(* Logix 5000 project; controller RSL5k_18_Template_noLib Emulate 5570 rev 32.11; software revision 32.02; part 7 of 16 *)
(* tags used below, declared in another part *)
   Inp_CascSP : ALIAS FOR Wrk_PIDE.SPCascade;   // Setpoint in Cascade, Independent PV in Ratio (PVEU)
   Inp_CVPrev : REAL;   // Previous scan CV (CVEU)
   Inp_OvrdCmd : DINT;   // Loop Mode command in Override: 0=None, 1=Man, 2=Auto, 3=Casc, 4=Norm, 5=Start SP Ramp, 6=Stop SP Ramp
   Inp_OvrdSP : REAL;   // Loop Auto Setpoint (SP) in Override (PVEU)
   Inp_OvrdCV : REAL;   // Loop Manual Output (CV) in Override (CVEU)
   Inp_OvrdSPTarget : REAL;   // Override Setpoint Target for SP Ramping ('wizard') (PVEU)
   Inp_OvrdSPRoCLimInc : REAL;   // Override Setting for Setpoint Positive Rate of Change Limit (PVEU/sec)
   Inp_OvrdSPRoCLimDec : REAL;   // Override Setting for Setpoint Negative Rate of Change Limit (PVEU/sec)
   Inp_Reset : BOOL;   // 1=Reset latched Alarms
   Cfg_HasRatio : ALIAS FOR Wrk_PIDE.UseRatio;   // 1=Casc Loop Mode is Ratio, 0=Casc Loop Mode is Cascade
   Cfg_HasCasc : ALIAS FOR Wrk_PIDE.AllowCasRat;   // 1=Enable the loop to be placed into cascade/ratio mode
   Cfg_HasAuto : BOOL;   // 1=Enable the loop to be placed into automatic mode
   Cfg_HasMan : BOOL;   // 1=Enable the loop to be placed into manual mode
   Cfg_LockLM : BOOL;   // Lock Loop Mode: 0=not locked, 1=locked in Normal mode (see Cfg_NormLM)
   Cfg_HasMoreObj : BOOL;   // 1=Tells HMI an object with more info is available
   Cfg_OvrdIntlk : BOOL;   // 1=Override ignores Bypassable Intlk; 0=always use Intlk
   Cfg_NormLM : DINT;   // Normal Loop Mode 0=Disable Normal selection, 1=Man, 2=Auto, 3=Casc
   Cfg_PwrupLM : DINT;   // Powerup Loop Mode 0=No change (last), 1=Man (w/ CV), 2=Auto (w/ SP), 3=Casc, 4=Normal
   Cfg_SPFailSPAct : DINT;   // SP Fail Setpoint Action: 1=hold last good, 2=use Cfg_IntlkSP, 3=set SP to curr. PV
   Cfg_PVFailCVAct : DINT;   // PV Fail CV Action: 1=hold last good, 2=use Cfg_IntlkCV
   Cfg_CVFailCVAct : DINT;   // CV Fail CV Action: 1=hold last good, 2=use Cfg_IntlkCV
   Cfg_PVDecPlcs : DINT;   // Number of decimal places for display of PV / SP
   Cfg_CVDecPlcs : DINT;   // Number of decimal places for display of CV
   Cfg_MaxSPRoCInc : REAL;   // Maximum allowed Setpoint Positive Rate of Change Limit (PVEU/sec)
   Cfg_MaxSPRoCDec : REAL;   // Maximum allowed Setpoint Negative Rate of Change Limit (PVEU/sec)
   Cfg_CVEUMin : REAL;   // CV Engineering Units Minimum Value (CVEU)
   Cfg_CVEUMax : REAL;   // CV Engineering Units Maximum Value (CVEU)
   Cfg_PGain : ALIAS FOR Wrk_PIDE.PGain;   // Proportional (independent) or Loop (dependent) Gain (unitless)
   Cfg_IGain : ALIAS FOR Wrk_PIDE.IGain;   // Integral Gain (1/min independent or min/repeat dependent)
   Cfg_DGain : ALIAS FOR Wrk_PIDE.DGain;   // Derivative Gain (min)
   Cfg_ZCDB : ALIAS FOR Wrk_PIDE.ZCDeadband;   // Normal Zero Crossing Deadband (PVEU)
   Cfg_CVRoCLim : REAL;   // CV Rate of Change Limit (CVEU/sec)
   Cfg_IntlkCV : REAL;   // CV Value to use with Interlock / Bad Value CV action (CVEU)
   Cfg_PwrupSP : REAL;   // Loop SP on powerup, used if Cfg_PwrupLM = 1 (Manual) or 2 (Auto) (PVEU)
   Cfg_PwrupCV : REAL;   // Loop CV on powerup, used if Cfg_PwrupLM <> 0 (none) (CVEU)
   Cfg_HiHiDevDB : REAL;   // High-High Devation Status Deadband (PVEU)
   Cfg_HiDevDB : REAL;   // High Devation Status Deadband (PVEU)
   Cfg_LoDevDB : REAL;   // Low Devation Status Deadband (PVEU)
   Cfg_LoLoDevDB : REAL;   // Low-Low Devation Status Deadband (PVEU)
   Cfg_OperKeep : SINT;   // Oper keeps control: .0=Loop Mode .1=CV .2=SP, .3=Ratio
   Cfg_ProgKeep : SINT;   // Prog keeps control: .0=Loop Mode .1=CV .2=SP, .3=Ratio
   Cfg_ExtKeep : SINT;   // Ext keeps control: .0=Loop Mode .1=CV .2=SP, .3=Ratio
   PSet_SP : REAL;   // Program Setting for Setpoint (loop Auto) (PVEU)
   PSet_SPRoCLimInc : REAL;   // Program Setting for Setpoint Rate of Change Limit Increasing (PVEU/sec)
   PSet_SPRoCLimDec : REAL;   // Program Setting for Setpoint Rate of Change Limit Decreasing (PVEU/sec)
   PSet_SPTarget : REAL;   // Program Setting for Setpoint Ramp Target (endpoint, for ramp wizard) (PVEU)
   PSet_CV : REAL;   // Program Setting for Controlled Variable (loop Manual) (CVEU)
   PSet_Owner : DINT;   // Program Owner Request ID (non-zero) or Release (zero)
   XSet_SP : REAL;   // External Setting for Setpoint (loop Auto) (PVEU)
   XSet_SPRoCLimInc : REAL;   // External Setting for Setpoint Rate of Change Limit Increasing (PVEU/sec)
   XSet_SPRoCLimDec : REAL;   // External Setting for Setpoint Rate of Change Limit Decreasing (PVEU/sec)
   XSet_SPTarget : REAL;   // External Setting for Setpoint Ramp Target (endpoint, for ramp wizard) (PVEU)
   XSet_CV : REAL;   // External Setting for Controlled Variable (loop Manual) (CVEU)
   PCmd_Casc : BOOL;   // Program Command to select Cascade / Ratio Loop Mode
   PCmd_Auto : BOOL;   // Program Command to select Automatic Loop Mode
   PCmd_Man : BOOL;   // Program Command to select Manual Loop Mode
   PCmd_NormLM : BOOL;   // Operator Command to select Normal Loop Mode (see Cfg_NormLM)
   PCmd_SPRampStart : BOOL;   // Program Command to initiate SP ramping
   PCmd_SPRampStop : BOOL;   // Program Command to stop SP ramping
   PCmd_Reset : BOOL;   // Program Command to Reset all Alarms requiring Reset
   XCmd_Casc : BOOL;   // External Command to select Cascade / Ratio control
   XCmd_Auto : BOOL;   // External Command to select Automatic control
   XCmd_Man : BOOL;   // External Command to select Manual control
   XCmd_NormLM : BOOL;   // External Command to select Normal Loop Mode (see Cfg_NormLM)
   XCmd_SPRampStart : BOOL;   // External Command to initiate SP ramping
   XCmd_SPRampStop : BOOL;   // External Command to stop SP ramping
   XCmd_Reset : BOOL;   // External Command to Reset all Alarms requiring Reset
   Val_Ratio : ALIAS FOR Wrk_PIDE.Ratio;   // Value of Loop Ratio (unitless)
   Val_SPSet : REAL;   // Value of selected SP (before clamping and ramping) (PVEU)
   Val_SP : ALIAS FOR Wrk_PIDE.SP;   // Value of SP being used (after ramping and clamping (PVEU)
   Val_SPTarget : REAL;   // Accepted Setting for Setpoint Ramp Target (endpoint, for ramp wizard) (PVEU)
   Val_CVSet : REAL;   // Value of selected CV (before clamping and ramping) (CVEU)
   Val_CVOut : REAL;   // Value of CV Output (after ramping and clamping (CVEU)
   Val_Owner : DINT;   // Current Object Owner ID (0=not owned)
   Sts_PVBad : BOOL;   // 1=PV Value, comms, quality or EU Limitis Bad
   Sts_Bypass : BOOL;   // 1=Bypassable Interlocks are Bypassed
   Sts_BypActive : BOOL;   // 1=Bypassing Active (Bypassed or Maintenance)
   Nrdy_OoS : BOOL;   // 1=Device Not Ready: Out of Service
   Sts_MaintByp : BOOL;   // 1=Device has a Maintenance Bypass function active
   Err_CVEU : BOOL;   // 1=Error in Config: CV EU Max/Min Invalid
   Sts_OoS : ALIAS FOR CmdSrc.Sts_OoS;
   Sts_Maint : ALIAS FOR CmdSrc.Sts_Maint;
   Sts_Ovrd : ALIAS FOR CmdSrc.Sts_Ovrd;
   Sts_Ext : ALIAS FOR CmdSrc.Sts_Ext;
   Sts_Prog : ALIAS FOR CmdSrc.Sts_Prog;
   Sts_Oper : ALIAS FOR CmdSrc.Sts_Oper;
   Sts_RdyAck : BOOL;   // 1=An alarm is ready to be acknowledged
   P_PIDE : BOOL;   // Unique Parameter Name for auto - discovery
   CmdSrc : P_CmdSrc;   // Control / Command Source Selection
   Fail : P_Alarm;   // Loop (SP, PV or CV) Failure Alarm
   IntlkTrip : P_Alarm;   // Interlock Trip Alarm
   Cfg_Tag : STRING_20;   // Tagname displayed on HMI
   Cfg_Label : STRING_20;   // Label for graphic symbol displayed on HMI
   Cfg_Desc : STRING_40;   // Description displayed on HMI
   Wrk_Bypass : BOOL;   // Internal Bypassable Interlocks are Bypassed flag
   Cfg_PVEU : STRING_8;   // PV / Setpoint Engineering Units displayed on HMI
   Wrk_ProgKeepONS : SINT;   // Program Keep one-shot stores
   Wrk_OperKeepONS : SINT;   // Operator Keep one-shot stores
   Wrk_ExtKeepONS : SINT;   // External Keep one-shot stores
   LoLoDev : P_Alarm;   // Low-Low Deviation Alarm
   LoDev : P_Alarm;   // Low Deviation Alarm
   HiDev : P_Alarm;   // High Deviation Alarm
   HiHiDev : P_Alarm;   // High-High Deviation Alarm
   Cfg_CVEU : STRING_8;   // CV Engineering Units displayed on HMI
   Wrk_Casc : BOOL;   // Internal Loop Mode latch: Cascade selected
   Wrk_Auto : BOOL;   // Internal Loop Mode latch: 1=Auto selected
   Wrk_Man : BOOL;   // Internal Loop Mode latch: Manual selected
   HMI_Type : STRING_16;   // Must contain AOI name, used for HMI and Information S/W
   Wrk_IntlkTripShed : BOOL;   // Shed Latch for Interlock Not OK
   Wrk_PVFailShed : BOOL;   // Shed Latch for PV Failure
   Wrk_SPFailShed : BOOL;   // Shed Latch for SP Failure
   Wrk_CVFailShed : BOOL;   // Shed Latch for CV Failure
   Wrk_ShedMan : BOOL;   // A shed condition is forcing Loop Mode to Manual
   Wrk_ShedAuto : BOOL;   // A shed condition is forcing Loop Mode to Auto or Manual
   Cfg_CVNavTag : STRING_NavTag;   // Tagname for destination of CV Navigation button
   Cfg_PVNavTag : STRING_NavTag;   // Tagname for destination of PV Navigation button
   Cfg_CascSPNavTag : STRING_NavTag;   // Tagname for destination of Cascade SP Navigation button
   HMI_Lib : STRING_12;   // Display Library for Faceplate call-up
   Wrk_PIDE : PID_ENHANCED;   // Built-in controller PID algorithm
   Cfg_Area : STRING_Area;   // Process Area for security
   Wrk_Autotune : PIDE_AUTOTUNE;   // Autotune tag associated with built-in PID algorithm
   HMI_HasAutotune : BOOL;   // 1=P_PIDE_Only AOI has been modified to include Autotune par. on PIDE block
   OCmd_ResetAckAll : BOOL;   // Operator Command to Reset all Alarms and latched Shed conditions
   OCmd_Reset : BOOL;   // Operator Command to Reset all Alarms requiring Reset
   MCmd_Check : BOOL;   // Maintenance Command to Check (not bypass) all Interlocks
   MCmd_Bypass : BOOL;   // Maintenance Command to Bypass all Bypassable Interlocks
   OCmd_SPRampStop : BOOL;   // Operator Command to stop SP ramping
   OCmd_SPRampStart : BOOL;   // Operator Command to initiate SP ramping
   OCmd_NormLM : BOOL;   // Operator Command to select Normal Loop Mode (see Cfg_NormLM)
   OCmd_Man : BOOL;   // Operator Command to select Manual control
   OCmd_Auto : BOOL;   // Operator Command to select Automatic control
   OCmd_Casc : BOOL;   // Operator Command to select Cascade / Ratio control
   OSet_CV : REAL;   // Operator Setting for Controlled Variable (loop Manual) (CVEU)
   OSet_SPTarget : REAL;   // Operator Setting for Setpoint Ramp Target (endpoint, for ramp wizard) (PVEU)
   OSet_SPRoCLimDec : REAL;   // Operator Setting for Setpoint Rate of Change Limit Decreasing (PVEU/sec)
   OSet_SPRoCLimInc : REAL;   // Operator Setting for Setpoint Rate of Change Limit Increasing (PVEU/sec)
   OSet_SP : REAL;   // Operator Setting for Setpoint (loop Auto) (PVEU)
   Wrk_ExtHas : SINT;   // External owns: .0=LM, .1=CV, .2=SP, .3=Ratio
   Wrk_ProgHas : SINT;   // Program owns: .0=LM, .1=CV, .2=SP, .3=Ratio
   Wrk_OperHas : SINT;   // Operator owns: .0=LM, .1=CV, .2=SP, .3=Ratio
   MRdy_Check : BOOL;   // 1=Ready for MCmd_Check (enables HMI button)
   MRdy_Bypass : BOOL;   // 1=Ready for MCmd_Bypass (enables HMI button)
   Wrk_Init : BOOL;   // 1=AOI has been initialized
(* P_PIDE, continued *)

ROUTINE Logic   (* ladder *)
// Normal Scan: control PID Loop
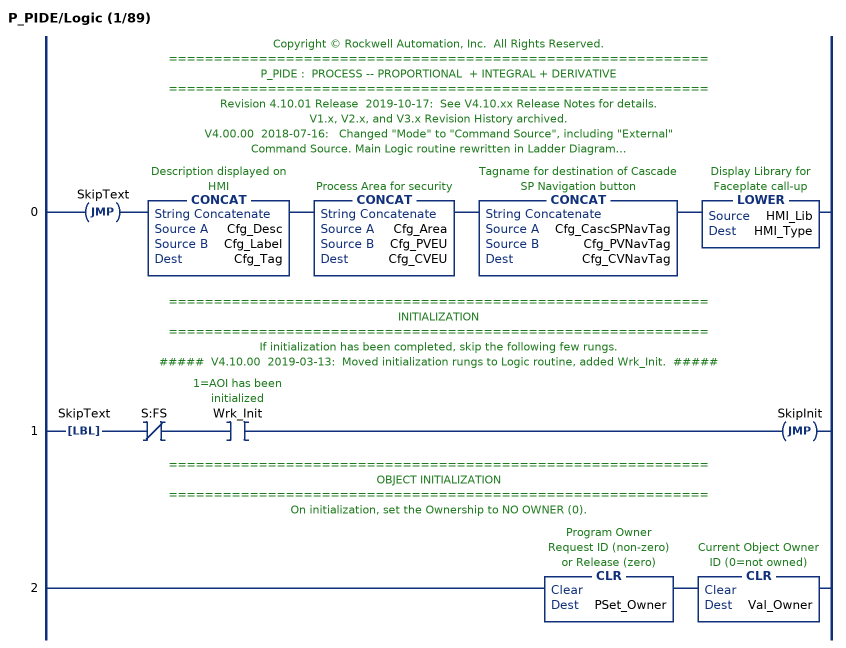
   // Copyright © Rockwell Automation, Inc.  All Rights Reserved.
   // ============================================================
   // P_PIDE :  PROCESS -- PROPORTIONAL  + INTEGRAL + DERIVATIVE
   // ============================================================
   // Revision 4.10.01 Release  2019-10-17:  See V4.10.xx Release Notes for details.
   // V1.x, V2.x, and V3.x Revision History archived.
   // V4.00.00  2018-07-16:   Changed "Mode" to "Command Source", including "External"
   // Command Source. Main Logic routine rewritten in Ladder Diagram.
   // Changed Inf_ items to HMI_, and added Cfg_Area for security.
   // Added notify and unack count rollup for connected objects.
   // Deleted Cfg_PCmdClear.  All Program Commands are now self-clearing.
   // Aligned ready bit naming with command bit names.
   // All OCmds/MCmds and ORdys/MRdys are now Local Tags.
   // Added Sts_RdyAck and Sts_ResetReqd for use by external objects.
   // Added SP Ramping and Ramp Wizard.  Added capability to have CV range
   // other than 0 to 100%.  Added Shed options.  Added Normal Loop Mode, locking
   // of Loop Mode. Added Oper / Prog / Ext "Keep" for Loop Mode, CV, SP, Ratio.
   // V4.00.01  2018-08-29:  Updated Override Command Source operation and description of Inp_OvrdCmd.
   // V4.00.02  2018-12-10:  Modified handling of CV I/O Fault, CV Fail and Shed configurations.
   // Corrected handling of configured execution interval.
   // V4.10.00  2019-03-13:  Changed availability to use input availability from interlocks.
   // Corrected parameter and local tag descriptions and external access.
   // Added Cfg_HasMoreObj. Updated to P_CmdSrc V4.10.00.
   // Moved initialization rungs to Logic routine, added Wrk_Init to correct
   // locking of Autotune tag on online instance creation.
   // Corrected overwriting of user SP Rate of Change limits by SP ramp wizard.
   // V4.10.01  2019-10-17:  Corrected clamping of CV, Ratio settings in Manual.
   // Corrected determination of Val_CVSet based on CV Init status.
   // Corrected generation of Sts_PVBad. Corrected CV Rate of Change Limiting.
   // Modified Interlock function to use PIDE manual CV instead of override CV, to get CV ramping.
   // Corrected SP ramp increasing. Modified Cascade/Ratio logic to include SP rate limiting.
   // ============================================================
   // This Instruction is used to provide PID (Proportional + Integral +
   // Derivative) feedback loop control and provides:
   // *  Prog, Oper, and Ext entry of Auto loop mode Setpoint in Engineering Units
   // *  Prog, Oper, and Ext. entry of Setpoint Target and Ramp Time and
   // command to trigger a Setpoint Ramp ("SP Ramp Wizard")
   // *  Prog, Oper, and Ext. entry of Manual loop mode Controlled Variable (CV) in Percent
   // *  Clamping (in EU) and ramping (in EU/sec) of Setpoint at specified limits
   // (separate increase and decrease rate of change limits).
   // *  Clamping (in CVEU) and ramping (in CVEU/sec) of CV at specified limits
   // (separate increase and decrease rate of change limits).
   // *  CV in Engineering Units (CVEU) for use as Cascade Setpoint for a secondary loop\
   // plus scaling to Raw units for use with non-scaling I/O card
   // *  Reverse or Direct control action    *  Feedforward input
   // *  Velocity (difference) PID form (with inputs for "Previous" CV and FF)
   // *  Option for Derivative action based on change in Error or change in PV
   // *  Option for Proportional action based on Error or PV
   // *  Monitoring of Interlock conditions which cause output to shed
   // *  Configurable shed to HOLD or to configured SAFE value, shed SP to current PV.
   // *  Monitoring of I/O communication faults
   // *  Alarms for Interlock Trip, Loop Failure, High-High Deviation, High Deviation,
   // Low Deviation and Low-Low Deviation from Setpoint
   // *  Operation from Hand, Maintenance, Override, External Program and Operator command sources
   // *  Full loop control (Cascade, Auto with Setpoint, Manual with CV) available in Override
   // *  "Available" status for use by automation logic to know whether loop
   //       can be controlled via Program commands / settings from other objects.
   // Command Sources are arbitrated by a P_CmdSrc Add-On Instruction instance.
   // Command Sources: Operator, Program, External, Override, Maintenance,
   // Out of Service, Hand.  Alarms are provided by P_Alarm Add-On Instruction instances.
   // ============================================================
   // SHOW LOCAL STRINGS
   // ============================================================
   // The STRINGs containing the text associated with each instance of this
   // instruction cannot be Input or Output Parameters, because STRINGs are not
   //  'atomic' types. (Inputs and Outputs must be SINT, INT, DINT, REAL, or BOOL.)
   // In order to make it easier to find and configure these STRINGs, this rung
   // was added.  THE JMP (and the LBL on the following rung)
   // MUST NOT BE REMOVED!!!
   // To view the STRINGs, go to the instruction instance (in LD or FBD), RIGHT-click
   // to bring up the context menu and select "Open Instruction Logic".
   // This rung will appear with the STRING values for the selected instance.
   // You may double-click the STRING values here to modify them as well.
   // #####  V4.00.00  2018-07-16:  Added string for Cfg_Area, renamed Inf_* to HMI_*.  #####
   0: JMP(SkipText)CONCAT(Cfg_Desc,Cfg_Label,Cfg_Tag)CONCAT(Cfg_Area,Cfg_PVEU,Cfg_CVEU)CONCAT(Cfg_CascSPNavTag,Cfg_PVNavTag,Cfg_CVNavTag)LOWER(HMI_Lib,HMI_Type);
   // ============================================================
   // INITIALIZATION
   // ============================================================
   // If initialization has been completed, skip the following few rungs.
   // #####  V4.10.00  2019-03-13:  Moved initialization rungs to Logic routine, added Wrk_Init.  #####
   1: LBL(SkipText)XIO(S:FS)XIC(Wrk_Init)JMP(SkipInit);
   // ============================================================
   // OBJECT INITIALIZATION
   // ============================================================
   // On initialization, set the Ownership to NO OWNER (0).
   2: CLR(PSet_Owner)CLR(Val_Owner);
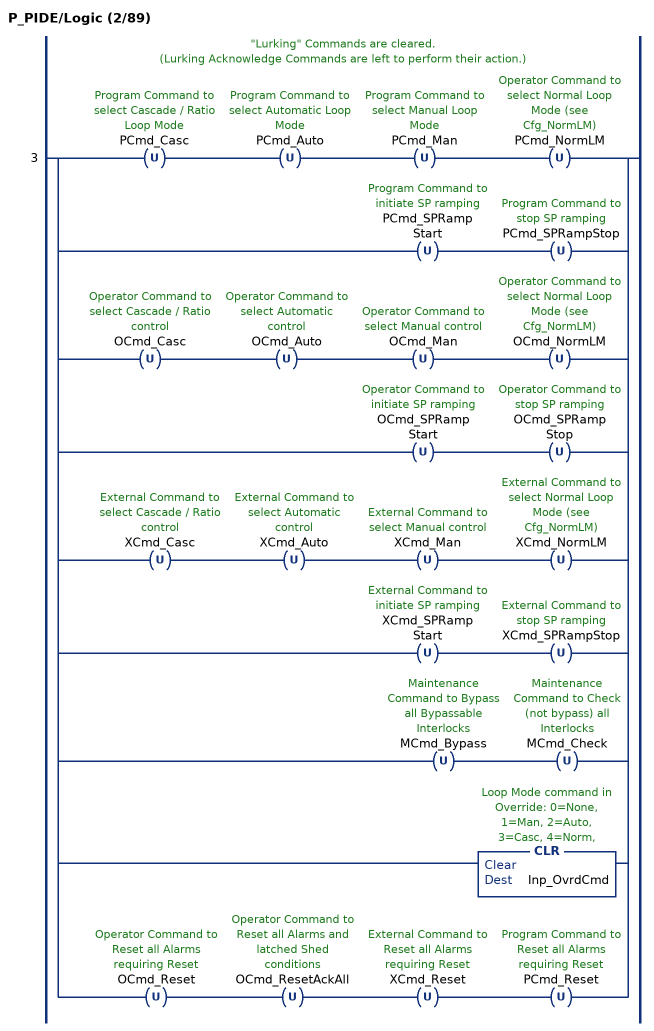
   // "Lurking" Commands are cleared.
   // (Lurking Acknowledge Commands are left to perform their action.)
   3: [OTU(PCmd_Casc) OTU(PCmd_Auto) OTU(PCmd_Man) OTU(PCmd_NormLM) ,OTU(PCmd_SPRampStart) OTU(PCmd_SPRampStop) ,OTU(OCmd_Casc) OTU(OCmd_Auto) OTU(OCmd_Man) OTU(OCmd_NormLM) ,OTU(OCmd_SPRampStart) OTU(OCmd_SPRampStop) ,OTU(XCmd_Casc) OTU(XCmd_Auto) OTU(XCmd_Man) OTU(XCmd_NormLM) ,OTU(XCmd_SPRampStart) OTU(XCmd_SPRampStop) ,OTU(MCmd_Bypass) OTU(MCmd_Check) ,CLR(Inp_OvrdCmd) ,OTU(OCmd_Reset) OTU(OCmd_ResetAckAll) OTU(XCmd_Reset) OTU(PCmd_Reset) ];
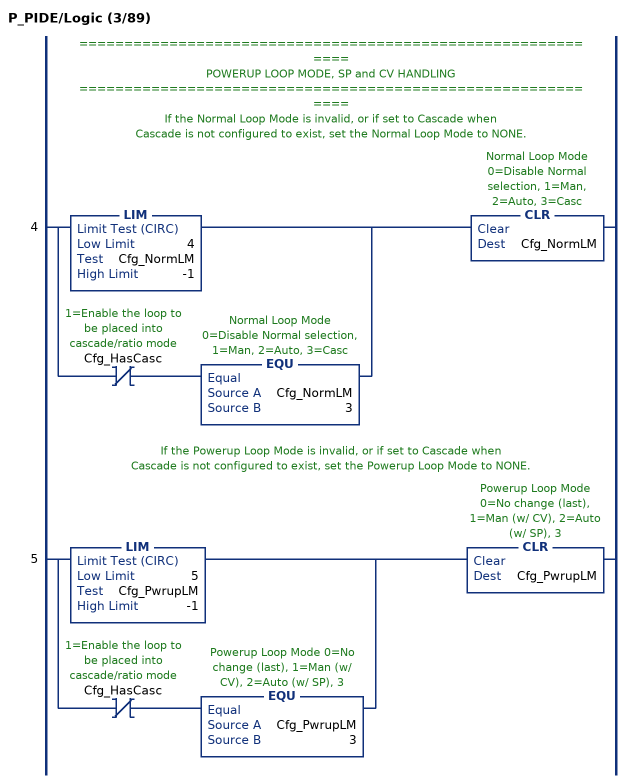
   // ============================================================
   // POWERUP LOOP MODE, SP and CV HANDLING
   // ============================================================
   // If the Normal Loop Mode is invalid, or if set to Cascade when
   // Cascade is not configured to exist, set the Normal Loop Mode to NONE.
   4: [LIM(4,Cfg_NormLM,-1) ,XIO(Cfg_HasCasc) EQU(Cfg_NormLM,3) ]CLR(Cfg_NormLM);
   // If the Powerup Loop Mode is invalid, or if set to Cascade when
   // Cascade is not configured to exist, set the Powerup Loop Mode to NONE.
   5: [LIM(5,Cfg_PwrupLM,-1) ,XIO(Cfg_HasCasc) EQU(Cfg_PwrupLM,3) ]CLR(Cfg_PwrupLM);
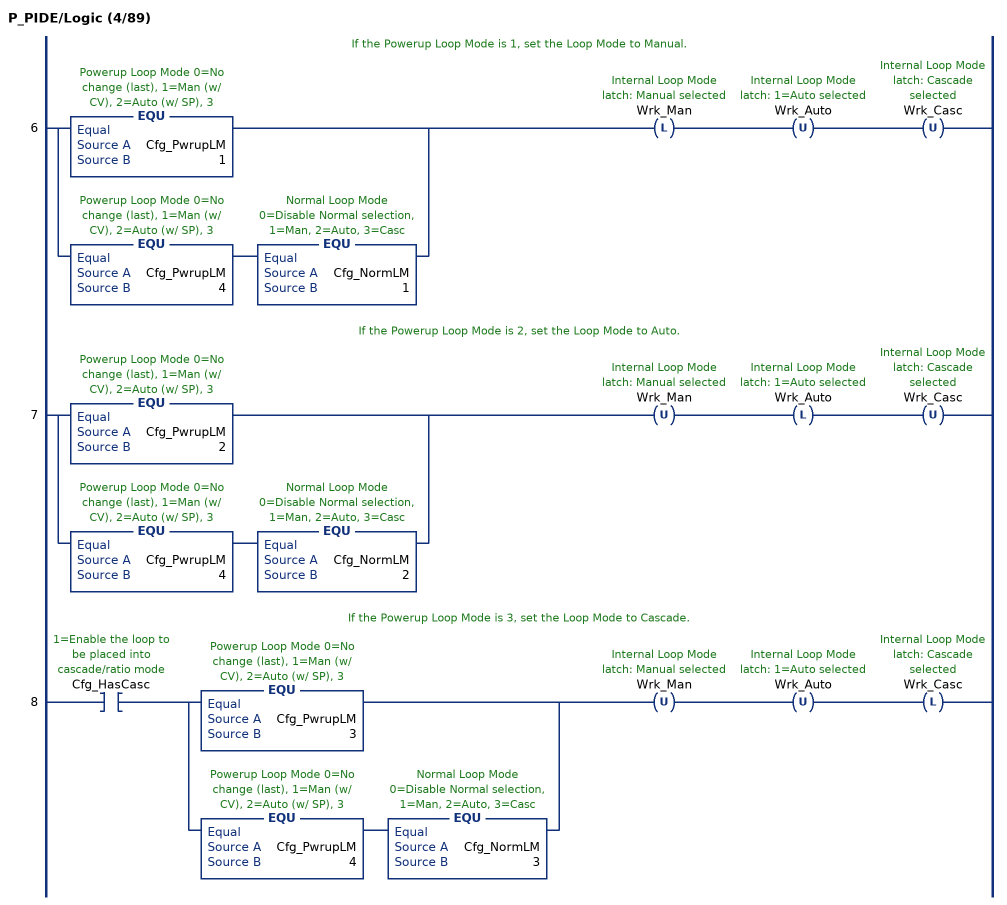
   // If the Powerup Loop Mode is 1, set the Loop Mode to Manual.
   6: [EQU(Cfg_PwrupLM,1) ,EQU(Cfg_PwrupLM,4) EQU(Cfg_NormLM,1) ]OTL(Wrk_Man)OTU(Wrk_Auto)OTU(Wrk_Casc);
   // If the Powerup Loop Mode is 2, set the Loop Mode to Auto.
   7: [EQU(Cfg_PwrupLM,2) ,EQU(Cfg_PwrupLM,4) EQU(Cfg_NormLM,2) ]OTU(Wrk_Man)OTL(Wrk_Auto)OTU(Wrk_Casc);
   // If the Powerup Loop Mode is 3, set the Loop Mode to Cascade.
   8: XIC(Cfg_HasCasc)[EQU(Cfg_PwrupLM,3) ,EQU(Cfg_PwrupLM,4) EQU(Cfg_NormLM,3) ]OTU(Wrk_Man)OTU(Wrk_Auto)OTL(Wrk_Casc);
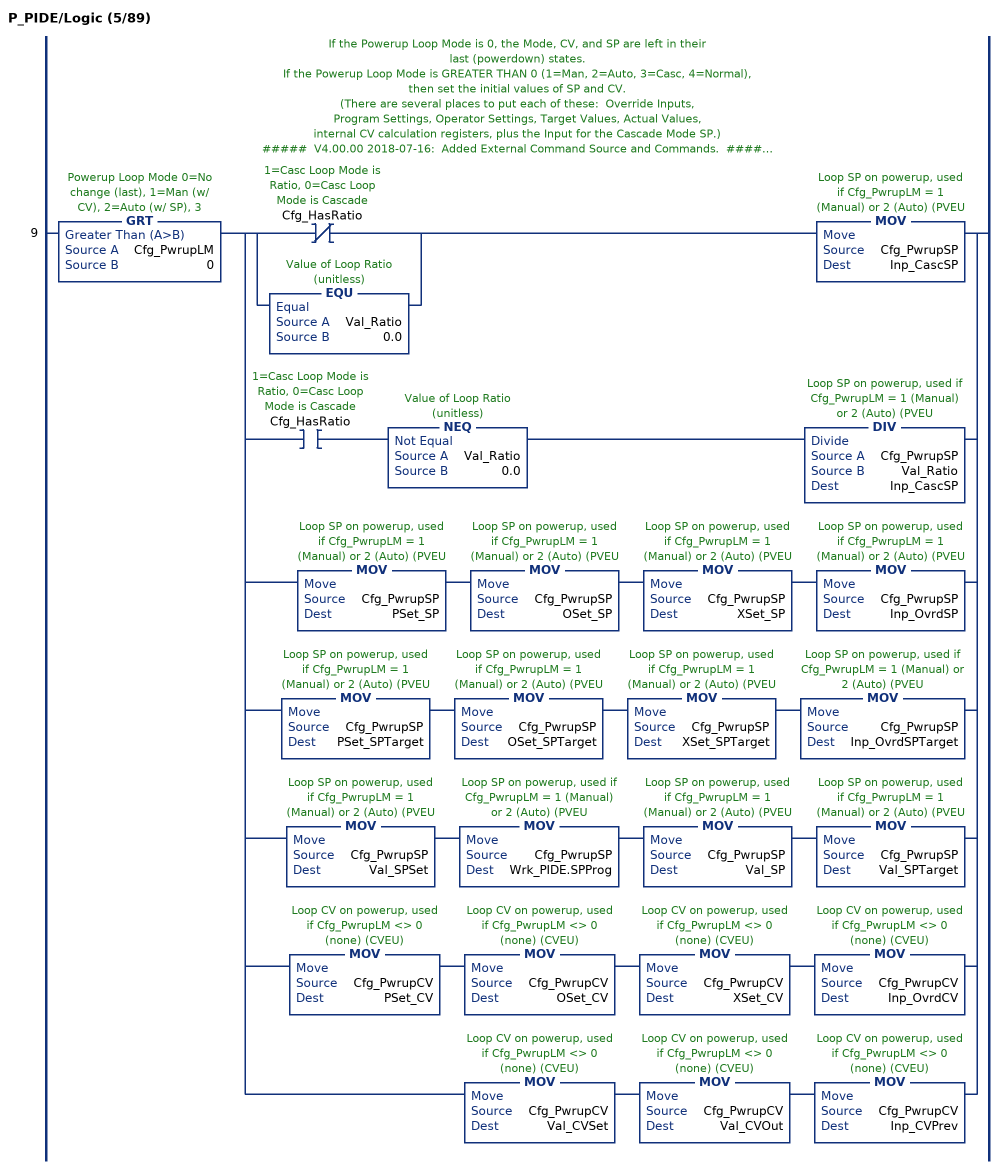
   // If the Powerup Loop Mode is 0, the Mode, CV, and SP are left in their
   // last (powerdown) states.
   // If the Powerup Loop Mode is GREATER THAN 0 (1=Man, 2=Auto, 3=Casc, 4=Normal),
   // then set the initial values of SP and CV.
   // (There are several places to put each of these:  Override Inputs,
   // Program Settings, Operator Settings, Target Values, Actual Values,
   // internal CV calculation registers, plus the Input for the Cascade Mode SP.)
   // #####  V4.00.00 2018-07-16:  Added External Command Source and Commands.  #####
   // #####  V4.00.02  2018-12-10:  Modified handling of CV Init, CV I/O Fault, and Powerup CV.  #####
   9: GRT(Cfg_PwrupLM,0)[[[XIO(Cfg_HasRatio) ,EQU(Val_Ratio,0.0) ] MOV(Cfg_PwrupSP,Inp_CascSP) ,XIC(Cfg_HasRatio) NEQ(Val_Ratio,0.0) DIV(Cfg_PwrupSP,Val_Ratio,Inp_CascSP) ] ,MOV(Cfg_PwrupSP,PSet_SP) MOV(Cfg_PwrupSP,OSet_SP) MOV(Cfg_PwrupSP,XSet_SP) MOV(Cfg_PwrupSP,Inp_OvrdSP) ,MOV(Cfg_PwrupSP,PSet_SPTarget) MOV(Cfg_PwrupSP,OSet_SPTarget) MOV(Cfg_PwrupSP,XSet_SPTarget) MOV(Cfg_PwrupSP,Inp_OvrdSPTarget) ,MOV(Cfg_PwrupSP,Val_SPSet) MOV(Cfg_PwrupSP,Wrk_PIDE.SPProg) MOV(Cfg_PwrupSP,Val_SP) MOV(Cfg_PwrupSP,Val_SPTarget) ,MOV(Cfg_PwrupCV,PSet_CV) MOV(Cfg_PwrupCV,OSet_CV) MOV(Cfg_PwrupCV,XSet_CV) MOV(Cfg_PwrupCV,Inp_OvrdCV) ,MOV(Cfg_PwrupCV,Val_CVSet) MOV(Cfg_PwrupCV,Val_CVOut) MOV(Cfg_PwrupCV,Inp_CVPrev) ];
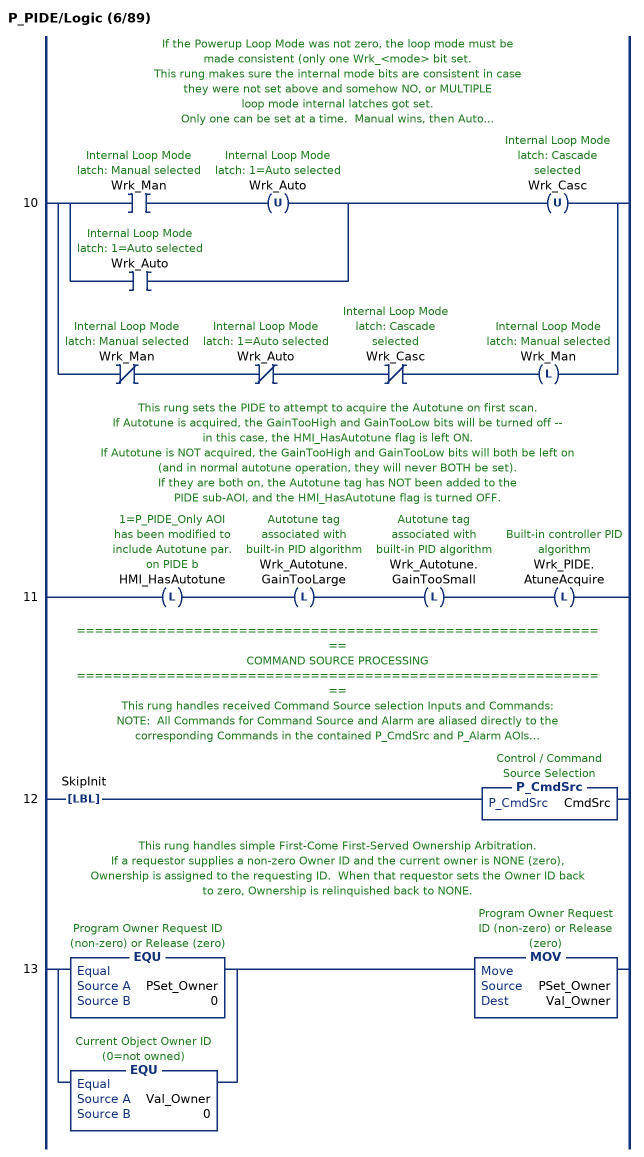
   // If the Powerup Loop Mode was not zero, the loop mode must be
   // made consistent (only one Wrk_<mode> bit set.
   // This rung makes sure the internal mode bits are consistent in case
   // they were not set above and somehow NO, or MULTIPLE
   // loop mode internal latches got set.
   // Only one can be set at a time.  Manual wins, then Auto...
   10: [[XIC(Wrk_Man) OTU(Wrk_Auto) ,XIC(Wrk_Auto) ] OTU(Wrk_Casc) ,XIO(Wrk_Man) XIO(Wrk_Auto) XIO(Wrk_Casc) OTL(Wrk_Man) ];
   // This rung sets the PIDE to attempt to acquire the Autotune on first scan.
   // If Autotune is acquired, the GainTooHigh and GainTooLow bits will be turned off --
   // in this case, the HMI_HasAutotune flag is left ON.
   // If Autotune is NOT acquired, the GainTooHigh and GainTooLow bits will both be left on
   // (and in normal autotune operation, they will never BOTH be set).
   // If they are both on, the Autotune tag has NOT been added to the
   // PIDE sub-AOI, and the HMI_HasAutotune flag is turned OFF.
   11: OTL(HMI_HasAutotune)OTL(Wrk_Autotune.GainTooLarge)OTL(Wrk_Autotune.GainTooSmall)OTL(Wrk_PIDE.AtuneAcquire);
   // ============================================================
   // COMMAND SOURCE PROCESSING
   // ============================================================
   // This rung handles received Command Source selection Inputs and Commands:
   // NOTE:  All Commands for Command Source and Alarm are aliased directly to the
   // corresponding Commands in the contained P_CmdSrc and P_Alarm AOIs.
   // #####  V4.00.00  2018-07-16:  Changed P_Mode to P_CmdSrc.  #####
   // #####  V4.10.00  2019-03-13:  Moved initialization rungs to Logic routine, added Wrk_Init. Added LBL here.  #####
   12: LBL(SkipInit)P_CmdSrc(CmdSrc);
   // This rung handles simple First-Come First-Served Ownership Arbitration.
   // If a requestor supplies a non-zero Owner ID and the current owner is NONE (zero),
   // Ownership is assigned to the requesting ID.  When that requestor sets the Owner ID back
   // to zero, Ownership is relinquished back to NONE.
   13: [EQU(PSet_Owner,0) ,EQU(Val_Owner,0) ]MOV(PSet_Owner,Val_Owner);
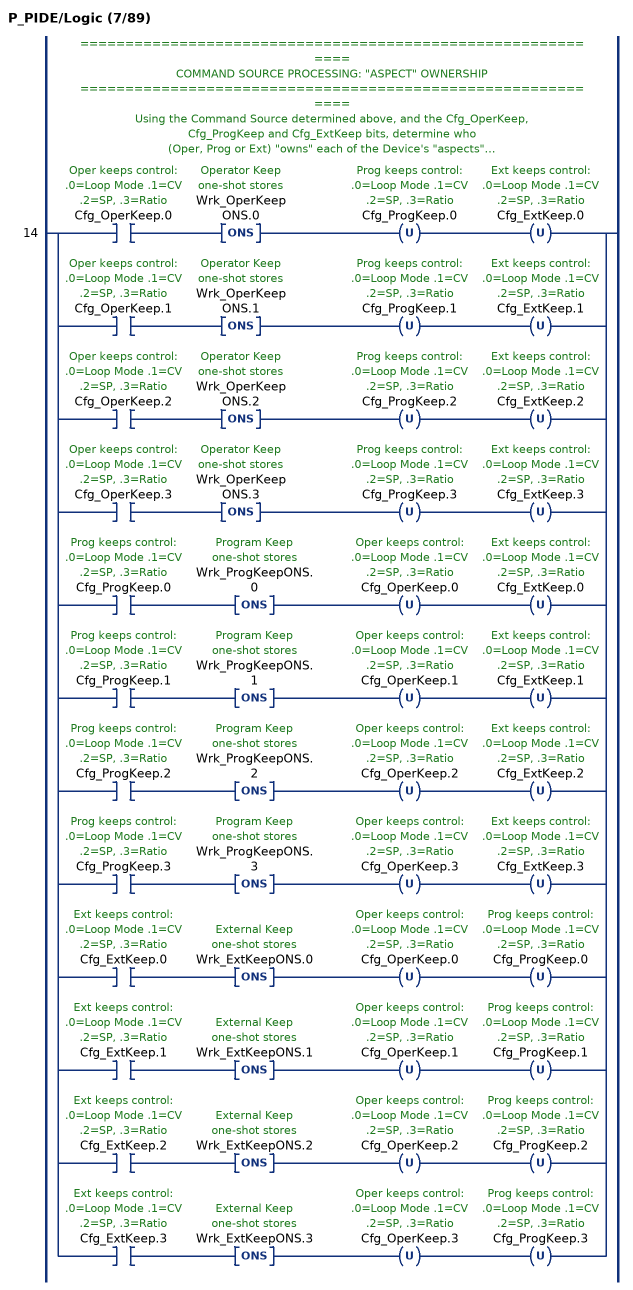
   // ============================================================
   // COMMAND SOURCE PROCESSING: "ASPECT" OWNERSHIP
   // ============================================================
   // Using the Command Source determined above, and the Cfg_OperKeep,
   // Cfg_ProgKeep and Cfg_ExtKeep bits, determine who
   // (Oper, Prog or Ext) "owns" each of the Device's "aspects":
   // Loop Mode (bit .0), Controlled Variable (CV, the output, bit .1),
   // Setpoint (SP, bit .2), and Ratio (bit .3).
   // The bits within Cfg_OperKeep, Cfg_ProgKeep and Cfg_ExtKeep determine
   // which "aspects" (sub-functions of this AOI) are retained by the Operator,
   // by the Program, or by the External command source when either of the
   // other command sources is selected.
   // All aspects (functions) may be "kept" (basically locking the Oper/Prog/Ext
   // selections, rendering the Command Source selection moot.
   // (You get to explain how it works to your operators!!!).
   // However, it is NOT allowed to have any given aspect "kept" by more than
   // one source.  This rung ensures that no aspect is "kept" by multiple sources.
   // #####  V4.00.00  2018-07-16:  Using P_CmdSrc, added External command source.  #####
   14: [XIC(Cfg_OperKeep.0) ONS(Wrk_OperKeepONS.0) OTU(Cfg_ProgKeep.0) OTU(Cfg_ExtKeep.0) ,XIC(Cfg_OperKeep.1) ONS(Wrk_OperKeepONS.1) OTU(Cfg_ProgKeep.1) OTU(Cfg_ExtKeep.1) ,XIC(Cfg_OperKeep.2) ONS(Wrk_OperKeepONS.2) OTU(Cfg_ProgKeep.2) OTU(Cfg_ExtKeep.2) ,XIC(Cfg_OperKeep.3) ONS(Wrk_OperKeepONS.3) OTU(Cfg_ProgKeep.3) OTU(Cfg_ExtKeep.3) ,XIC(Cfg_ProgKeep.0) ONS(Wrk_ProgKeepONS.0) OTU(Cfg_OperKeep.0) OTU(Cfg_ExtKeep.0) ,XIC(Cfg_ProgKeep.1) ONS(Wrk_ProgKeepONS.1) OTU(Cfg_OperKeep.1) OTU(Cfg_ExtKeep.1) ,XIC(Cfg_ProgKeep.2) ONS(Wrk_ProgKeepONS.2) OTU(Cfg_OperKeep.2) OTU(Cfg_ExtKeep.2) ,XIC(Cfg_ProgKeep.3) ONS(Wrk_ProgKeepONS.3) OTU(Cfg_OperKeep.3) OTU(Cfg_ExtKeep.3) ,XIC(Cfg_ExtKeep.0) ONS(Wrk_ExtKeepONS.0) OTU(Cfg_OperKeep.0) OTU(Cfg_ProgKeep.0) ,XIC(Cfg_ExtKeep.1) ONS(Wrk_ExtKeepONS.1) OTU(Cfg_OperKeep.1) OTU(Cfg_ProgKeep.1) ,XIC(Cfg_ExtKeep.2) ONS(Wrk_ExtKeepONS.2) OTU(Cfg_OperKeep.2) OTU(Cfg_ProgKeep.2) ,XIC(Cfg_ExtKeep.3) ONS(Wrk_ExtKeepONS.3) OTU(Cfg_OperKeep.3) OTU(Cfg_ProgKeep.3) ];
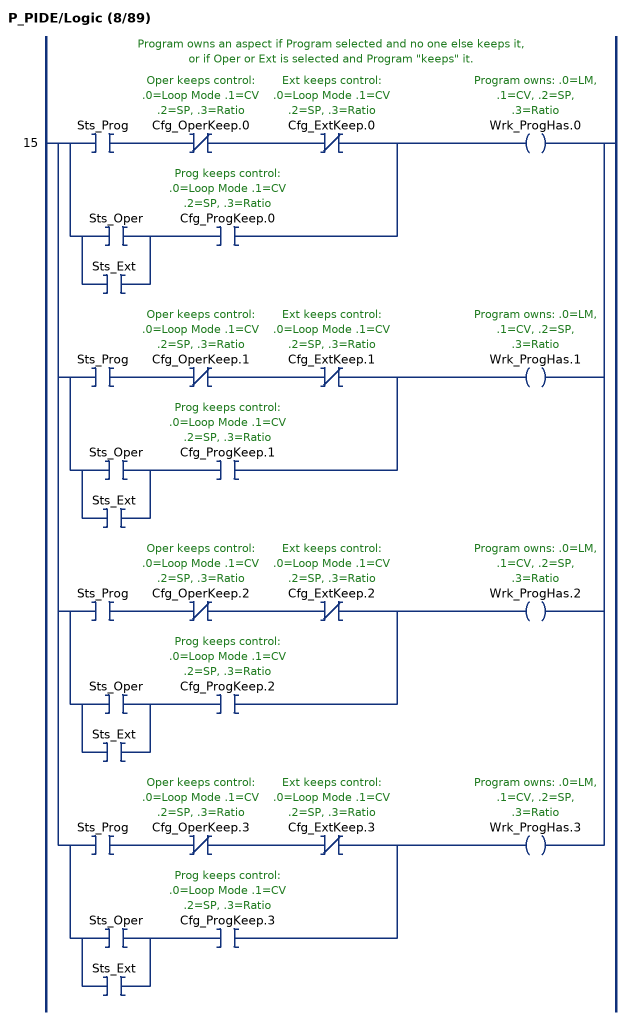
   // Program owns an aspect if Program selected and no one else keeps it,
   // or if Oper or Ext is selected and Program "keeps" it.
   15: [[XIC(Sts_Prog) XIO(Cfg_OperKeep.0) XIO(Cfg_ExtKeep.0) ,[XIC(Sts_Oper) ,XIC(Sts_Ext) ] XIC(Cfg_ProgKeep.0) ] OTE(Wrk_ProgHas.0) ,[XIC(Sts_Prog) XIO(Cfg_OperKeep.1) XIO(Cfg_ExtKeep.1) ,[XIC(Sts_Oper) ,XIC(Sts_Ext) ] XIC(Cfg_ProgKeep.1) ] OTE(Wrk_ProgHas.1) ,[XIC(Sts_Prog) XIO(Cfg_OperKeep.2) XIO(Cfg_ExtKeep.2) ,[XIC(Sts_Oper) ,XIC(Sts_Ext) ] XIC(Cfg_ProgKeep.2) ] OTE(Wrk_ProgHas.2) ,[XIC(Sts_Prog) XIO(Cfg_OperKeep.3) XIO(Cfg_ExtKeep.3) ,[XIC(Sts_Oper) ,XIC(Sts_Ext) ] XIC(Cfg_ProgKeep.3) ] OTE(Wrk_ProgHas.3) ];
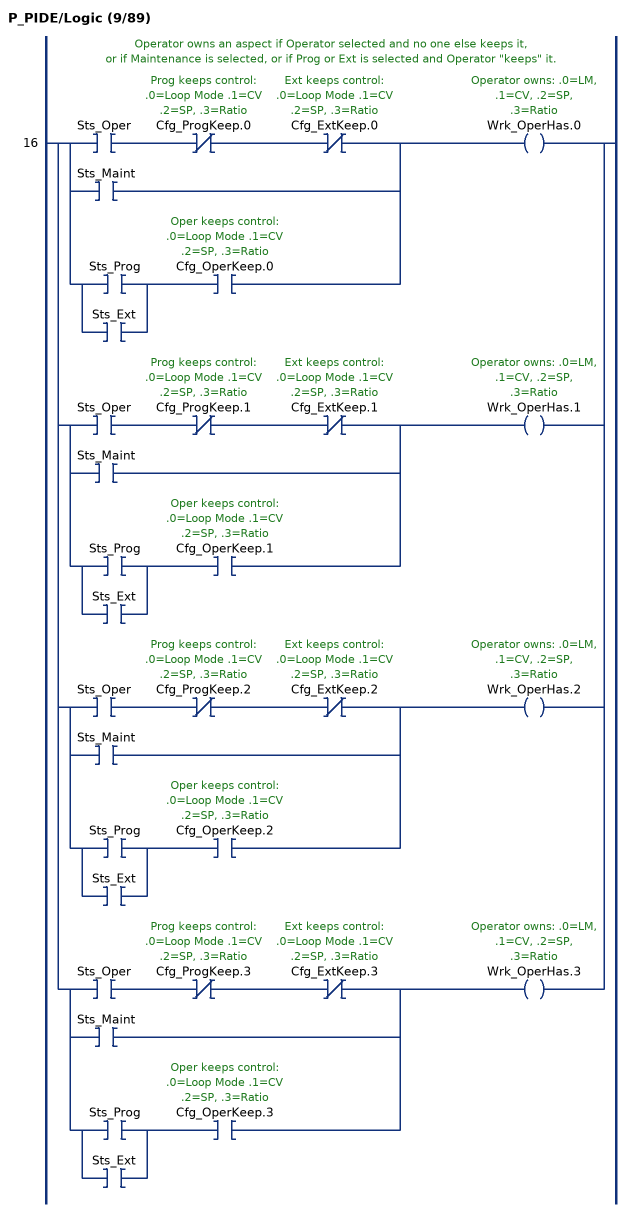
   // Operator owns an aspect if Operator selected and no one else keeps it,
   // or if Maintenance is selected, or if Prog or Ext is selected and Operator "keeps" it.
   16: [[XIC(Sts_Oper) XIO(Cfg_ProgKeep.0) XIO(Cfg_ExtKeep.0) ,XIC(Sts_Maint) ,[XIC(Sts_Prog) ,XIC(Sts_Ext) ] XIC(Cfg_OperKeep.0) ] OTE(Wrk_OperHas.0) ,[XIC(Sts_Oper) XIO(Cfg_ProgKeep.1) XIO(Cfg_ExtKeep.1) ,XIC(Sts_Maint) ,[XIC(Sts_Prog) ,XIC(Sts_Ext) ] XIC(Cfg_OperKeep.1) ] OTE(Wrk_OperHas.1) ,[XIC(Sts_Oper) XIO(Cfg_ProgKeep.2) XIO(Cfg_ExtKeep.2) ,XIC(Sts_Maint) ,[XIC(Sts_Prog) ,XIC(Sts_Ext) ] XIC(Cfg_OperKeep.2) ] OTE(Wrk_OperHas.2) ,[XIC(Sts_Oper) XIO(Cfg_ProgKeep.3) XIO(Cfg_ExtKeep.3) ,XIC(Sts_Maint) ,[XIC(Sts_Prog) ,XIC(Sts_Ext) ] XIC(Cfg_OperKeep.3) ] OTE(Wrk_OperHas.3) ];
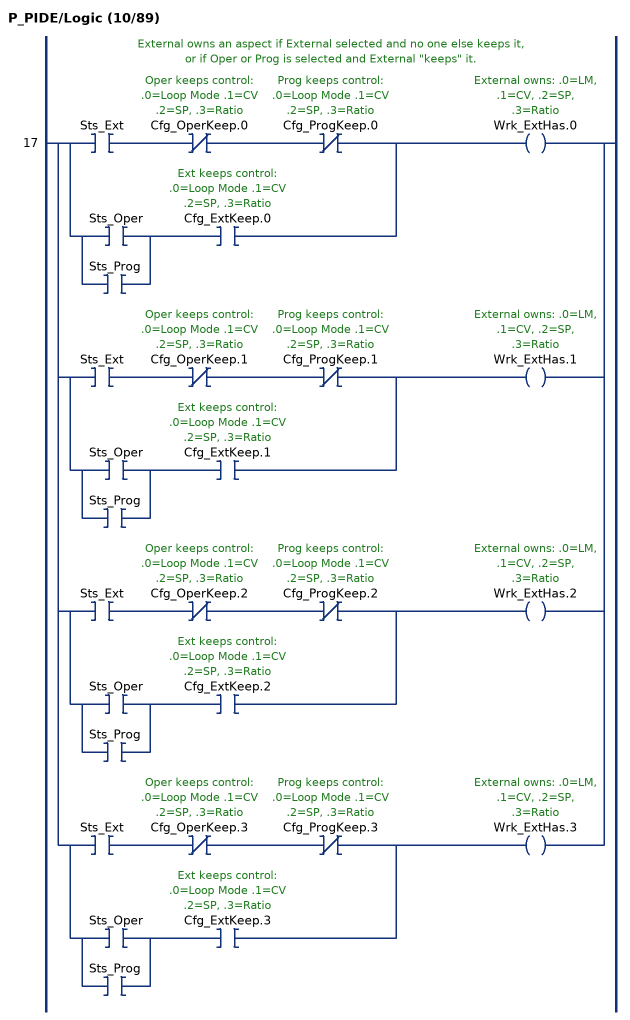
   // External owns an aspect if External selected and no one else keeps it,
   // or if Oper or Prog is selected and External "keeps" it.
   17: [[XIC(Sts_Ext) XIO(Cfg_OperKeep.0) XIO(Cfg_ProgKeep.0) ,[XIC(Sts_Oper) ,XIC(Sts_Prog) ] XIC(Cfg_ExtKeep.0) ] OTE(Wrk_ExtHas.0) ,[XIC(Sts_Ext) XIO(Cfg_OperKeep.1) XIO(Cfg_ProgKeep.1) ,[XIC(Sts_Oper) ,XIC(Sts_Prog) ] XIC(Cfg_ExtKeep.1) ] OTE(Wrk_ExtHas.1) ,[XIC(Sts_Ext) XIO(Cfg_OperKeep.2) XIO(Cfg_ProgKeep.2) ,[XIC(Sts_Oper) ,XIC(Sts_Prog) ] XIC(Cfg_ExtKeep.2) ] OTE(Wrk_ExtHas.2) ,[XIC(Sts_Ext) XIO(Cfg_OperKeep.3) XIO(Cfg_ProgKeep.3) ,[XIC(Sts_Oper) ,XIC(Sts_Prog) ] XIC(Cfg_ExtKeep.3) ] OTE(Wrk_ExtHas.3) ];
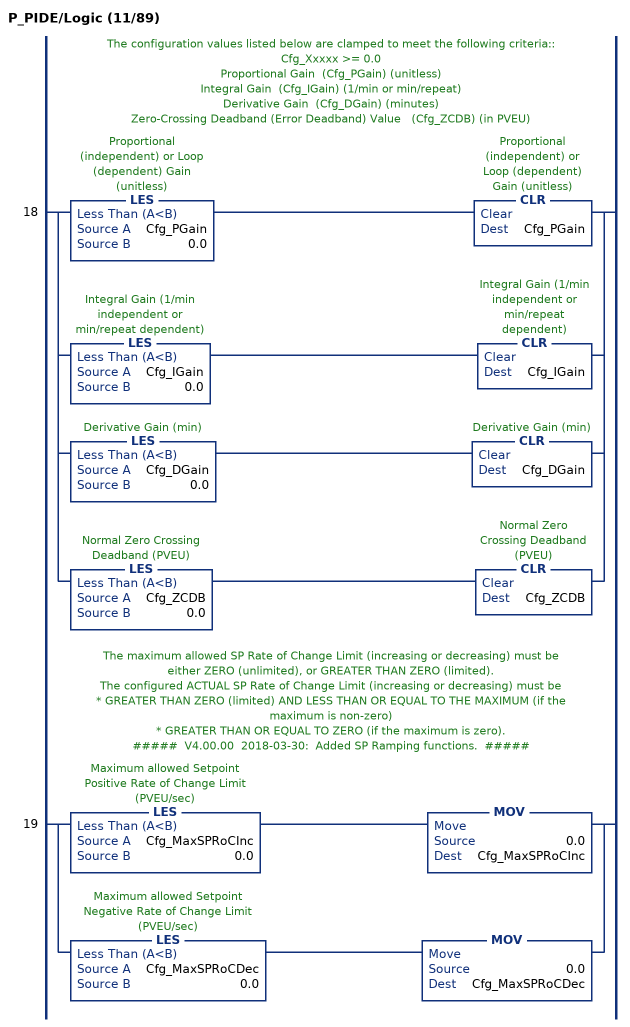
   // The configuration values listed below are clamped to meet the following criteria::
   // Cfg_Xxxxx >= 0.0
   // Proportional Gain  (Cfg_PGain) (unitless)
   //  Integral Gain  (Cfg_IGain) (1/min or min/repeat)
   // Derivative Gain  (Cfg_DGain) (minutes)
   // Zero-Crossing Deadband (Error Deadband) Value   (Cfg_ZCDB) (in PVEU)
   18: [LES(Cfg_PGain,0.0) CLR(Cfg_PGain) ,LES(Cfg_IGain,0.0) CLR(Cfg_IGain) ,LES(Cfg_DGain,0.0) CLR(Cfg_DGain) ,LES(Cfg_ZCDB,0.0) CLR(Cfg_ZCDB) ];
   // The maximum allowed SP Rate of Change Limit (increasing or decreasing) must be
   // either ZERO (unlimited), or GREATER THAN ZERO (limited).
   // The configured ACTUAL SP Rate of Change Limit (increasing or decreasing) must be
   // * GREATER THAN ZERO (limited) AND LESS THAN OR EQUAL TO THE MAXIMUM (if the maximum is non-zero)
   // * GREATER THAN OR EQUAL TO ZERO (if the maximum is zero).
   // #####  V4.00.00  2018-03-30:  Added SP Ramping functions.  #####
   19: [LES(Cfg_MaxSPRoCInc,0.0) MOV(0.0,Cfg_MaxSPRoCInc) ,LES(Cfg_MaxSPRoCDec,0.0) MOV(0.0,Cfg_MaxSPRoCDec) ];
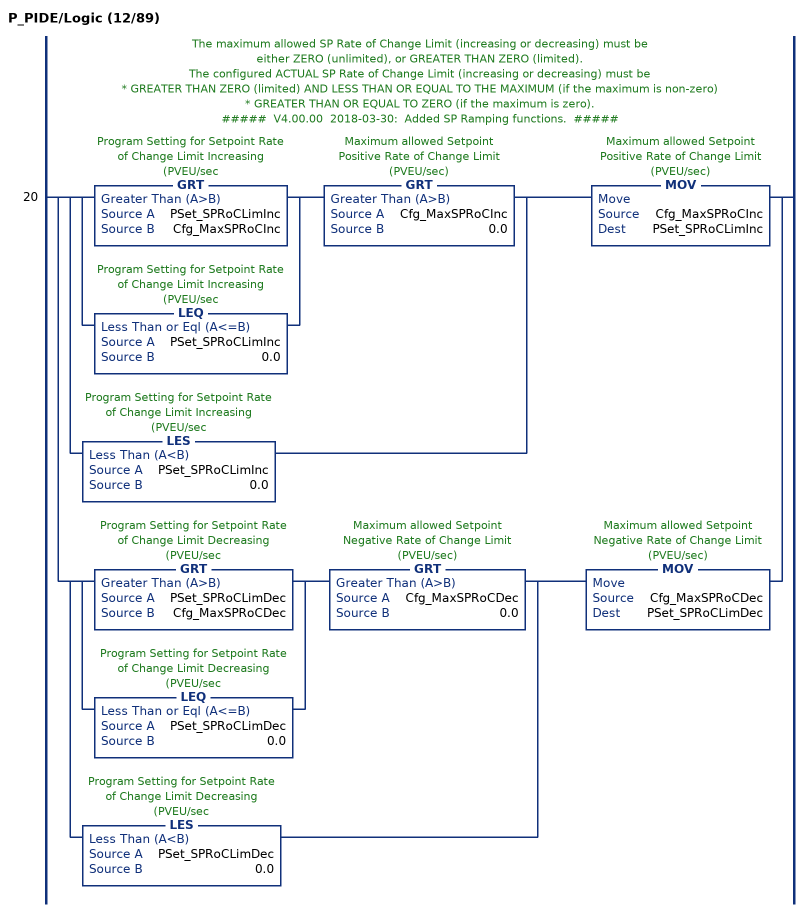
   // The maximum allowed SP Rate of Change Limit (increasing or decreasing) must be
   // either ZERO (unlimited), or GREATER THAN ZERO (limited).
   // The configured ACTUAL SP Rate of Change Limit (increasing or decreasing) must be
   // * GREATER THAN ZERO (limited) AND LESS THAN OR EQUAL TO THE MAXIMUM (if the maximum is non-zero)
   // * GREATER THAN OR EQUAL TO ZERO (if the maximum is zero).
   // #####  V4.00.00  2018-03-30:  Added SP Ramping functions.  #####
   20: [[[GRT(PSet_SPRoCLimInc,Cfg_MaxSPRoCInc) ,LEQ(PSet_SPRoCLimInc,0.0) ] GRT(Cfg_MaxSPRoCInc,0.0) ,LES(PSet_SPRoCLimInc,0.0) ] MOV(Cfg_MaxSPRoCInc,PSet_SPRoCLimInc) ,[[GRT(PSet_SPRoCLimDec,Cfg_MaxSPRoCDec) ,LEQ(PSet_SPRoCLimDec,0.0) ] GRT(Cfg_MaxSPRoCDec,0.0) ,LES(PSet_SPRoCLimDec,0.0) ] MOV(Cfg_MaxSPRoCDec,PSet_SPRoCLimDec) ];
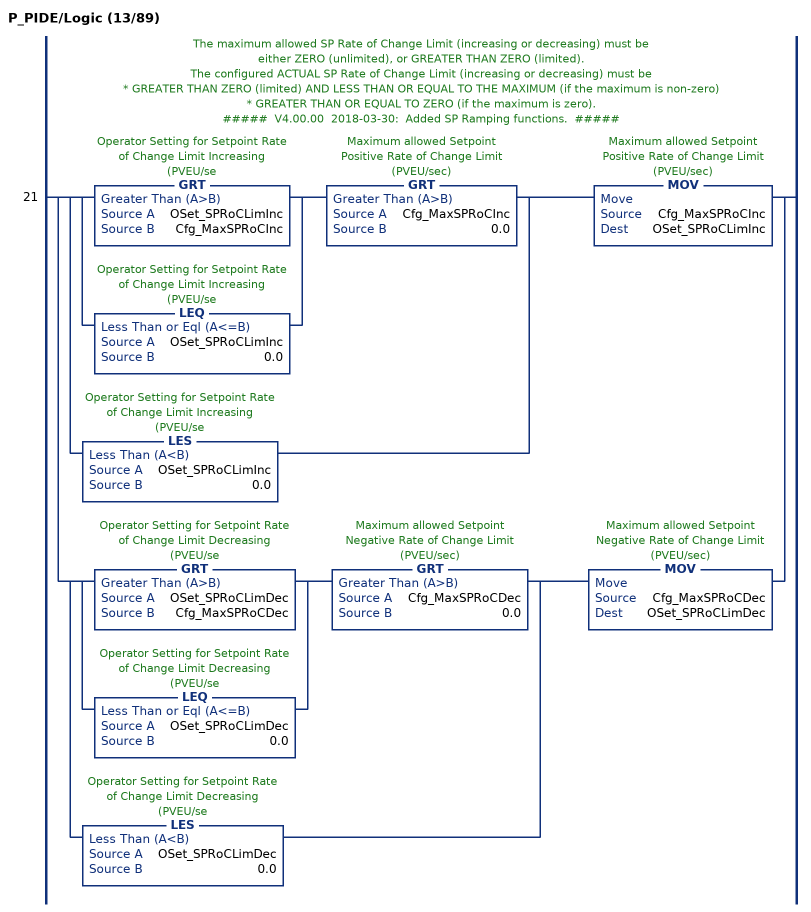
   // The maximum allowed SP Rate of Change Limit (increasing or decreasing) must be
   // either ZERO (unlimited), or GREATER THAN ZERO (limited).
   // The configured ACTUAL SP Rate of Change Limit (increasing or decreasing) must be
   // * GREATER THAN ZERO (limited) AND LESS THAN OR EQUAL TO THE MAXIMUM (if the maximum is non-zero)
   // * GREATER THAN OR EQUAL TO ZERO (if the maximum is zero).
   // #####  V4.00.00  2018-03-30:  Added SP Ramping functions.  #####
   21: [[[GRT(OSet_SPRoCLimInc,Cfg_MaxSPRoCInc) ,LEQ(OSet_SPRoCLimInc,0.0) ] GRT(Cfg_MaxSPRoCInc,0.0) ,LES(OSet_SPRoCLimInc,0.0) ] MOV(Cfg_MaxSPRoCInc,OSet_SPRoCLimInc) ,[[GRT(OSet_SPRoCLimDec,Cfg_MaxSPRoCDec) ,LEQ(OSet_SPRoCLimDec,0.0) ] GRT(Cfg_MaxSPRoCDec,0.0) ,LES(OSet_SPRoCLimDec,0.0) ] MOV(Cfg_MaxSPRoCDec,OSet_SPRoCLimDec) ];
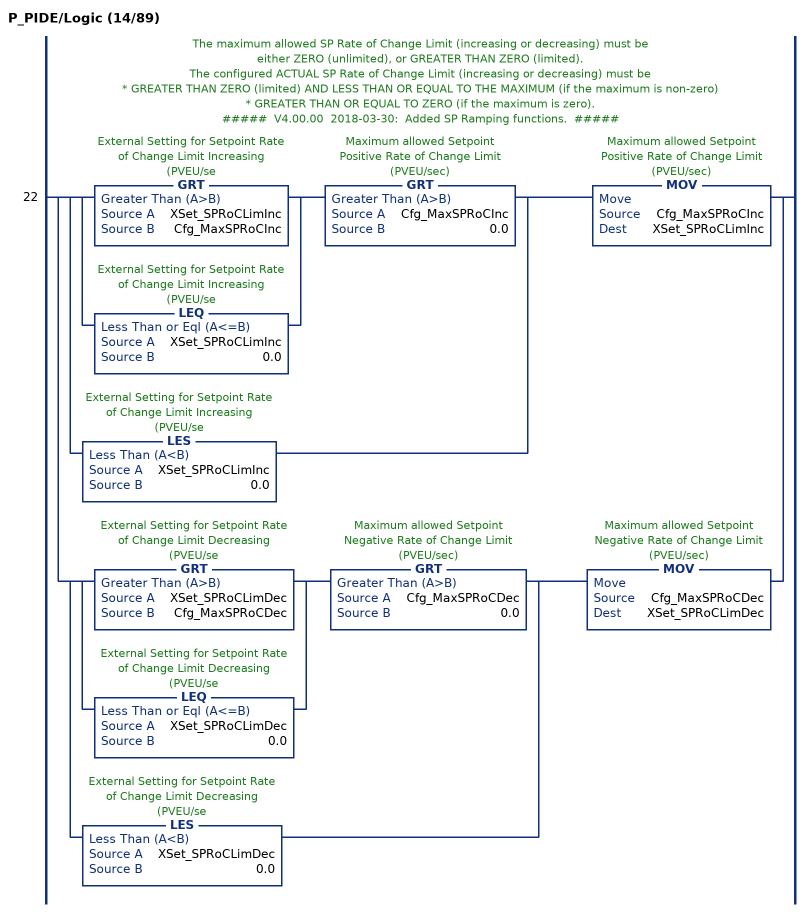
   // The maximum allowed SP Rate of Change Limit (increasing or decreasing) must be
   // either ZERO (unlimited), or GREATER THAN ZERO (limited).
   // The configured ACTUAL SP Rate of Change Limit (increasing or decreasing) must be
   // * GREATER THAN ZERO (limited) AND LESS THAN OR EQUAL TO THE MAXIMUM (if the maximum is non-zero)
   // * GREATER THAN OR EQUAL TO ZERO (if the maximum is zero).
   // #####  V4.00.00  2018-03-30:  Added SP Ramping functions.  #####
   22: [[[GRT(XSet_SPRoCLimInc,Cfg_MaxSPRoCInc) ,LEQ(XSet_SPRoCLimInc,0.0) ] GRT(Cfg_MaxSPRoCInc,0.0) ,LES(XSet_SPRoCLimInc,0.0) ] MOV(Cfg_MaxSPRoCInc,XSet_SPRoCLimInc) ,[[GRT(XSet_SPRoCLimDec,Cfg_MaxSPRoCDec) ,LEQ(XSet_SPRoCLimDec,0.0) ] GRT(Cfg_MaxSPRoCDec,0.0) ,LES(XSet_SPRoCLimDec,0.0) ] MOV(Cfg_MaxSPRoCDec,XSet_SPRoCLimDec) ];
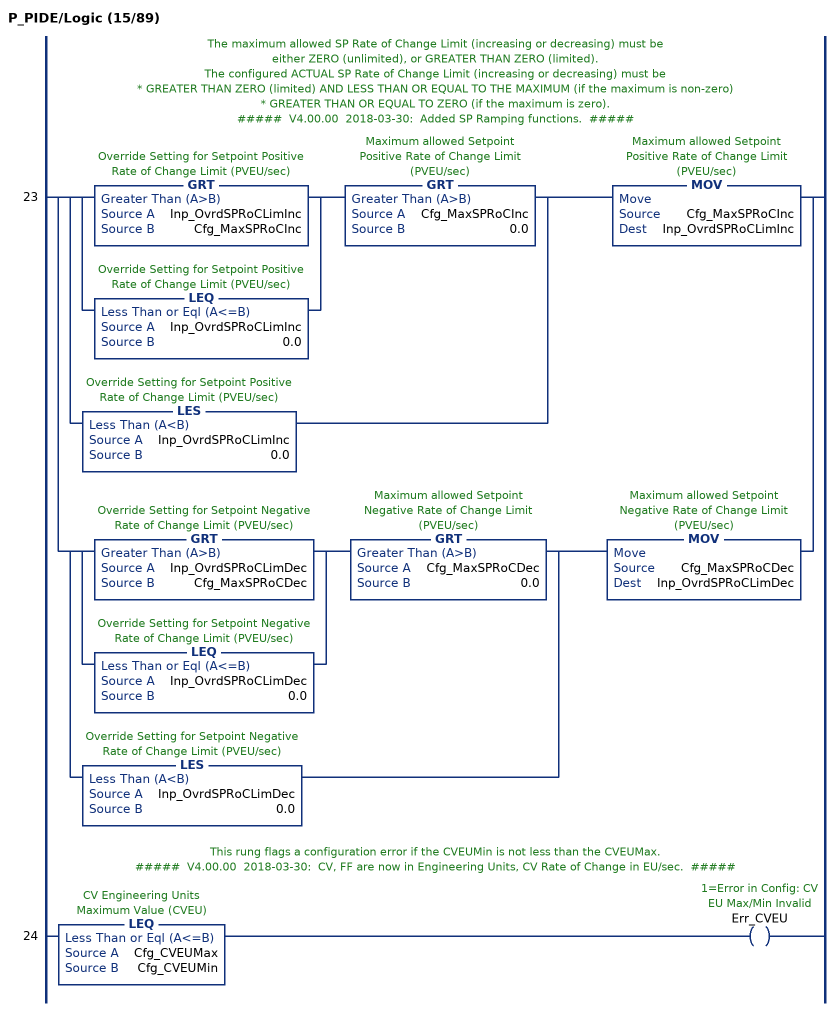
   // The maximum allowed SP Rate of Change Limit (increasing or decreasing) must be
   // either ZERO (unlimited), or GREATER THAN ZERO (limited).
   // The configured ACTUAL SP Rate of Change Limit (increasing or decreasing) must be
   // * GREATER THAN ZERO (limited) AND LESS THAN OR EQUAL TO THE MAXIMUM (if the maximum is non-zero)
   // * GREATER THAN OR EQUAL TO ZERO (if the maximum is zero).
   // #####  V4.00.00  2018-03-30:  Added SP Ramping functions.  #####
   23: [[[GRT(Inp_OvrdSPRoCLimInc,Cfg_MaxSPRoCInc) ,LEQ(Inp_OvrdSPRoCLimInc,0.0) ] GRT(Cfg_MaxSPRoCInc,0.0) ,LES(Inp_OvrdSPRoCLimInc,0.0) ] MOV(Cfg_MaxSPRoCInc,Inp_OvrdSPRoCLimInc) ,[[GRT(Inp_OvrdSPRoCLimDec,Cfg_MaxSPRoCDec) ,LEQ(Inp_OvrdSPRoCLimDec,0.0) ] GRT(Cfg_MaxSPRoCDec,0.0) ,LES(Inp_OvrdSPRoCLimDec,0.0) ] MOV(Cfg_MaxSPRoCDec,Inp_OvrdSPRoCLimDec) ];
   // This rung flags a configuration error if the CVEUMin is not less than the CVEUMax.
   // #####  V4.00.00  2018-03-30:  CV, FF are now in Engineering Units, CV Rate of Change in EU/sec.  #####
   24: LEQ(Cfg_CVEUMax,Cfg_CVEUMin)OTE(Err_CVEU);
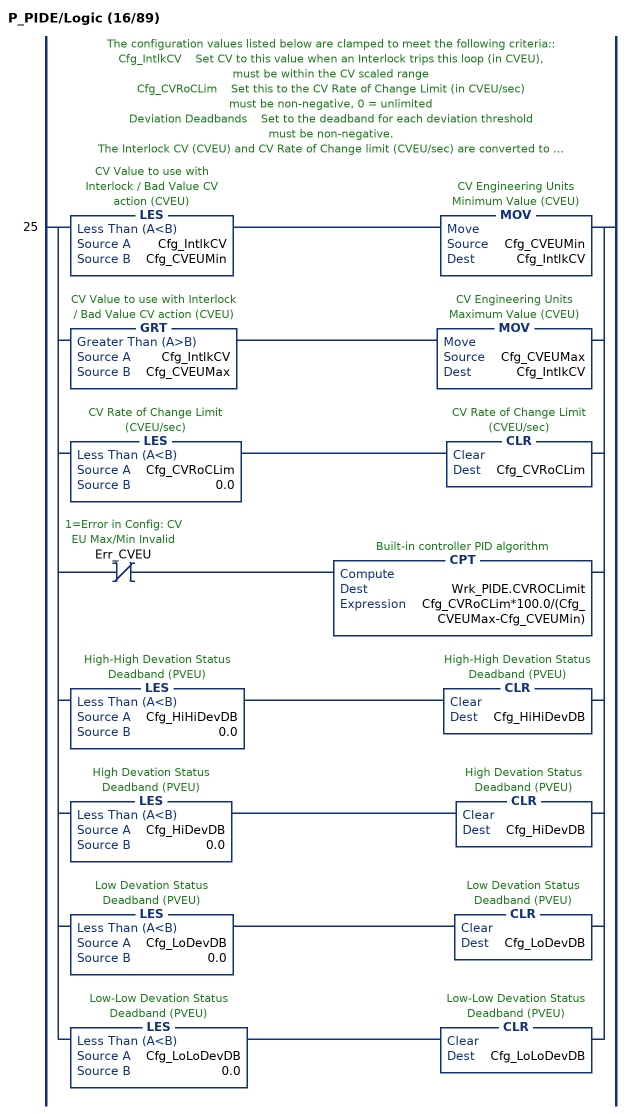
   // The configuration values listed below are clamped to meet the following criteria::
   // Cfg_IntlkCV    Set CV to this value when an Interlock trips this loop (in CVEU),
   // must be within the CV scaled range
   // Cfg_CVRoCLim    Set this to the CV Rate of Change Limit (in CVEU/sec)
   // must be non-negative, 0 = unlimited
   // Deviation Deadbands    Set to the deadband for each deviation threshold
   // must be non-negative.
   // The Interlock CV (CVEU) and CV Rate of Change limit (CVEU/sec) are converted to %
   // or %/sec and fed into the PIDE.
   // #####  V4.00.00  2018-03-30:  CV, FF are now in Engineering Units, CV Rate of Change in EU/sec.  #####
   25: [LES(Cfg_IntlkCV,Cfg_CVEUMin) MOV(Cfg_CVEUMin,Cfg_IntlkCV) ,GRT(Cfg_IntlkCV,Cfg_CVEUMax) MOV(Cfg_CVEUMax,Cfg_IntlkCV) ,LES(Cfg_CVRoCLim,0.0) CLR(Cfg_CVRoCLim) ,XIO(Err_CVEU) CPT(Wrk_PIDE.CVROCLimit,Cfg_CVRoCLim*100.0/(Cfg_CVEUMax-Cfg_CVEUMin)) ,LES(Cfg_HiHiDevDB,0.0) CLR(Cfg_HiHiDevDB) ,LES(Cfg_HiDevDB,0.0) CLR(Cfg_HiDevDB) ,LES(Cfg_LoDevDB,0.0) CLR(Cfg_LoDevDB) ,LES(Cfg_LoLoDevDB,0.0) CLR(Cfg_LoLoDevDB) ];
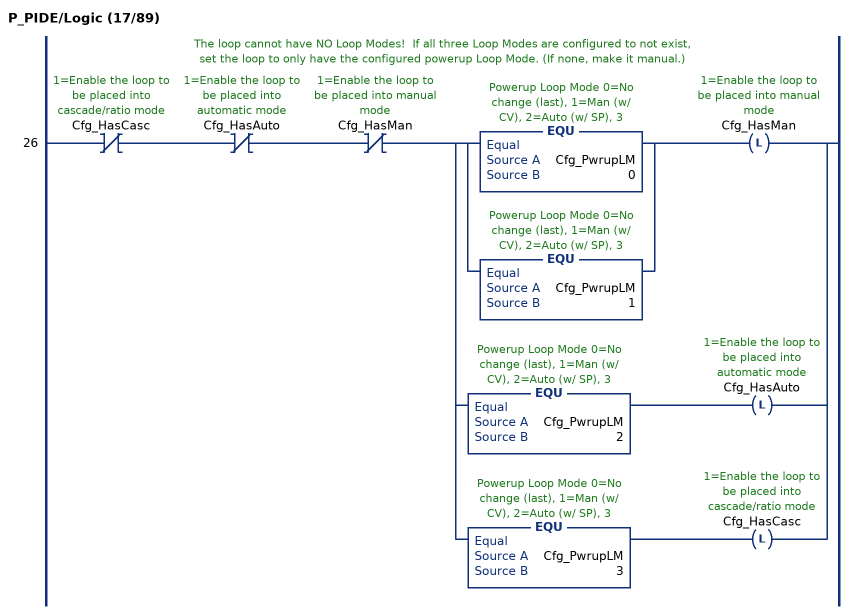
   // The loop cannot have NO Loop Modes!  If all three Loop Modes are configured to not exist,
   // set the loop to only have the configured powerup Loop Mode. (If none, make it manual.)
   26: XIO(Cfg_HasCasc)XIO(Cfg_HasAuto)XIO(Cfg_HasMan)[[EQU(Cfg_PwrupLM,0) ,EQU(Cfg_PwrupLM,1) ] OTL(Cfg_HasMan) ,EQU(Cfg_PwrupLM,2) OTL(Cfg_HasAuto) ,EQU(Cfg_PwrupLM,3) OTL(Cfg_HasCasc) ];
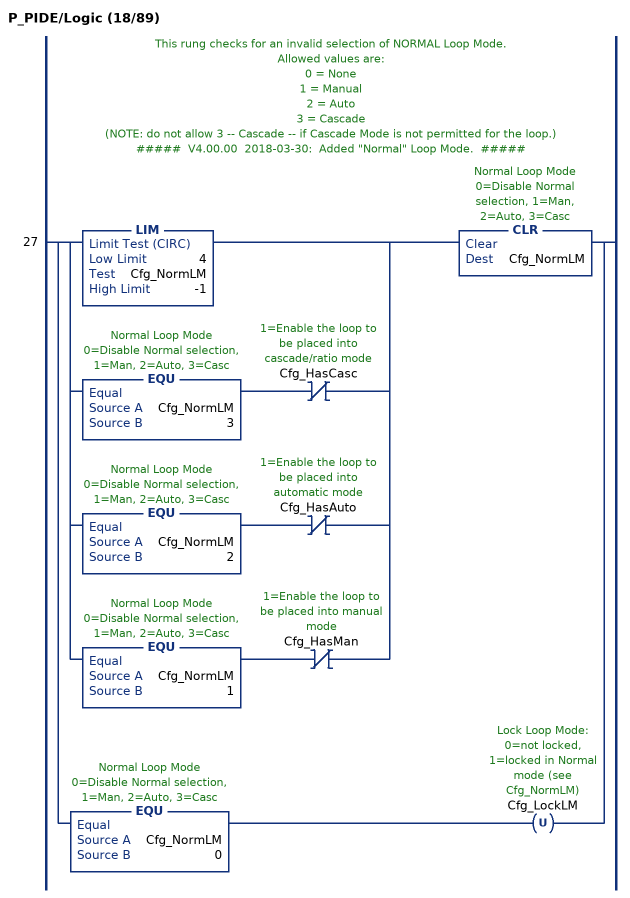
   // This rung checks for an invalid selection of NORMAL Loop Mode.
   // Allowed values are:
   // 0 = None
   // 1 = Manual
   // 2 = Auto
   // 3 = Cascade
   // (NOTE: do not allow 3 -- Cascade -- if Cascade Mode is not permitted for the loop.)
   // #####  V4.00.00  2018-03-30:  Added "Normal" Loop Mode.  #####
   27: [[LIM(4,Cfg_NormLM,-1) ,EQU(Cfg_NormLM,3) XIO(Cfg_HasCasc) ,EQU(Cfg_NormLM,2) XIO(Cfg_HasAuto) ,EQU(Cfg_NormLM,1) XIO(Cfg_HasMan) ] CLR(Cfg_NormLM) ,EQU(Cfg_NormLM,0) OTU(Cfg_LockLM) ];
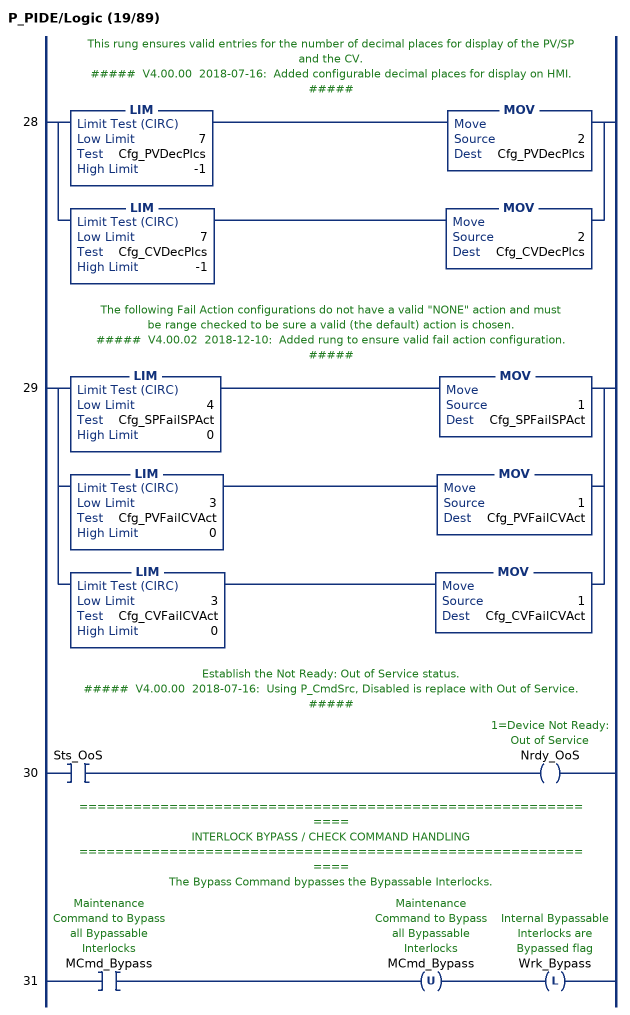
   // This rung ensures valid entries for the number of decimal places for display of the PV/SP and the CV.
   // #####  V4.00.00  2018-07-16:  Added configurable decimal places for display on HMI.  #####
   28: [LIM(7,Cfg_PVDecPlcs,-1) MOV(2,Cfg_PVDecPlcs) ,LIM(7,Cfg_CVDecPlcs,-1) MOV(2,Cfg_CVDecPlcs) ];
   // The following Fail Action configurations do not have a valid "NONE" action and must
   // be range checked to be sure a valid (the default) action is chosen.
   // #####  V4.00.02  2018-12-10:  Added rung to ensure valid fail action configuration.  #####
   29: [LIM(4,Cfg_SPFailSPAct,0) MOV(1,Cfg_SPFailSPAct) ,LIM(3,Cfg_PVFailCVAct,0) MOV(1,Cfg_PVFailCVAct) ,LIM(3,Cfg_CVFailCVAct,0) MOV(1,Cfg_CVFailCVAct) ];
   // Establish the Not Ready: Out of Service status.
   // #####  V4.00.00  2018-07-16:  Using P_CmdSrc, Disabled is replace with Out of Service.  #####
   30: XIC(Sts_OoS)OTE(Nrdy_OoS);
   // ============================================================
   // INTERLOCK BYPASS / CHECK COMMAND HANDLING
   // ============================================================
   // The Bypass Command bypasses the Bypassable Interlocks.
   31: XIC(MCmd_Bypass)OTU(MCmd_Bypass)OTL(Wrk_Bypass);
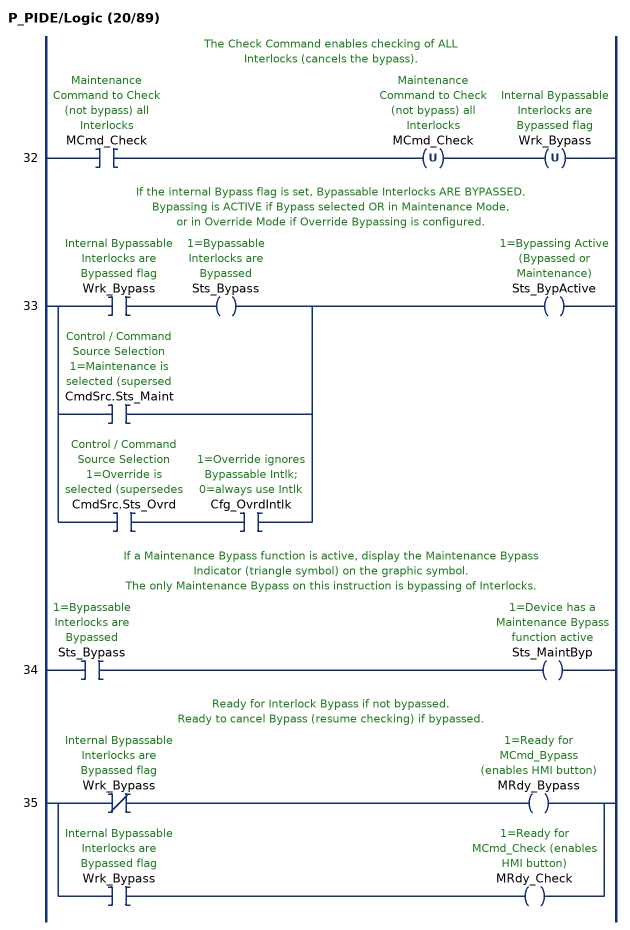
   // The Check Command enables checking of ALL
   // Interlocks (cancels the bypass).
   32: XIC(MCmd_Check)OTU(MCmd_Check)OTU(Wrk_Bypass);
   // If the internal Bypass flag is set, Bypassable Interlocks ARE BYPASSED.
   // Bypassing is ACTIVE if Bypass selected OR in Maintenance Mode,
   // or in Override Mode if Override Bypassing is configured.
   33: [XIC(Wrk_Bypass) OTE(Sts_Bypass) ,XIC(CmdSrc.Sts_Maint) ,XIC(CmdSrc.Sts_Ovrd) XIC(Cfg_OvrdIntlk) ]OTE(Sts_BypActive);
   // If a Maintenance Bypass function is active, display the Maintenance Bypass
   // Indicator (triangle symbol) on the graphic symbol.
   // The only Maintenance Bypass on this instruction is bypassing of Interlocks.
   34: XIC(Sts_Bypass)OTE(Sts_MaintByp);
   // Ready for Interlock Bypass if not bypassed.
   // Ready to cancel Bypass (resume checking) if bypassed.
   35: [XIO(Wrk_Bypass) OTE(MRdy_Bypass) ,XIC(Wrk_Bypass) OTE(MRdy_Check) ];
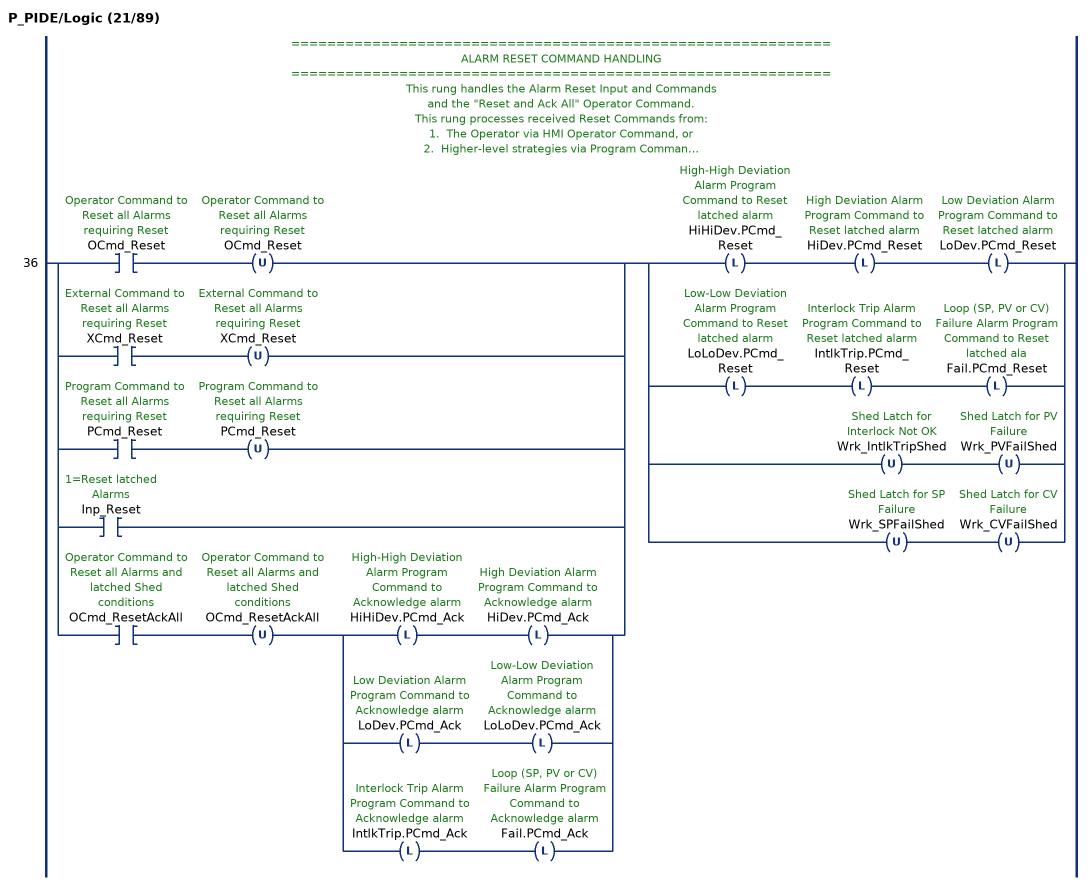
   // ============================================================
   // ALARM RESET COMMAND HANDLING
   // ============================================================
   // This rung handles the Alarm Reset Input and Commands
   // and the "Reset and Ack All" Operator Command.
   // This rung processes received Reset Commands from:
   // 1.  The Operator via HMI Operator Command, or
   // 2.  Higher-level strategies via Program Command
   // 3.  Pushbuttons or other block via Input
   // and forwards the Reset to ALL Alarms and latched Shed conditions.
   // #####  V4.00.00  2018-07-16:  Deleted Cfg_PCmdClear; all Program Commands are now self-clearing.  #####
   // #####  Changed P_Mode to P_CmdSrc. Added External Command Source and Commands.  #####
   36: [XIC(OCmd_Reset) OTU(OCmd_Reset) ,XIC(XCmd_Reset) OTU(XCmd_Reset) ,XIC(PCmd_Reset) OTU(PCmd_Reset) ,XIC(Inp_Reset) ,XIC(OCmd_ResetAckAll) OTU(OCmd_ResetAckAll) [OTL(HiHiDev.PCmd_Ack) OTL(HiDev.PCmd_Ack) ,OTL(LoDev.PCmd_Ack) OTL(LoLoDev.PCmd_Ack) ,OTL(IntlkTrip.PCmd_Ack) OTL(Fail.PCmd_Ack) ] ][OTL(HiHiDev.PCmd_Reset) OTL(HiDev.PCmd_Reset) OTL(LoDev.PCmd_Reset) ,OTL(LoLoDev.PCmd_Reset) OTL(IntlkTrip.PCmd_Reset) OTL(Fail.PCmd_Reset) ,OTU(Wrk_IntlkTripShed) OTU(Wrk_PVFailShed) ,OTU(Wrk_SPFailShed) OTU(Wrk_CVFailShed) ];
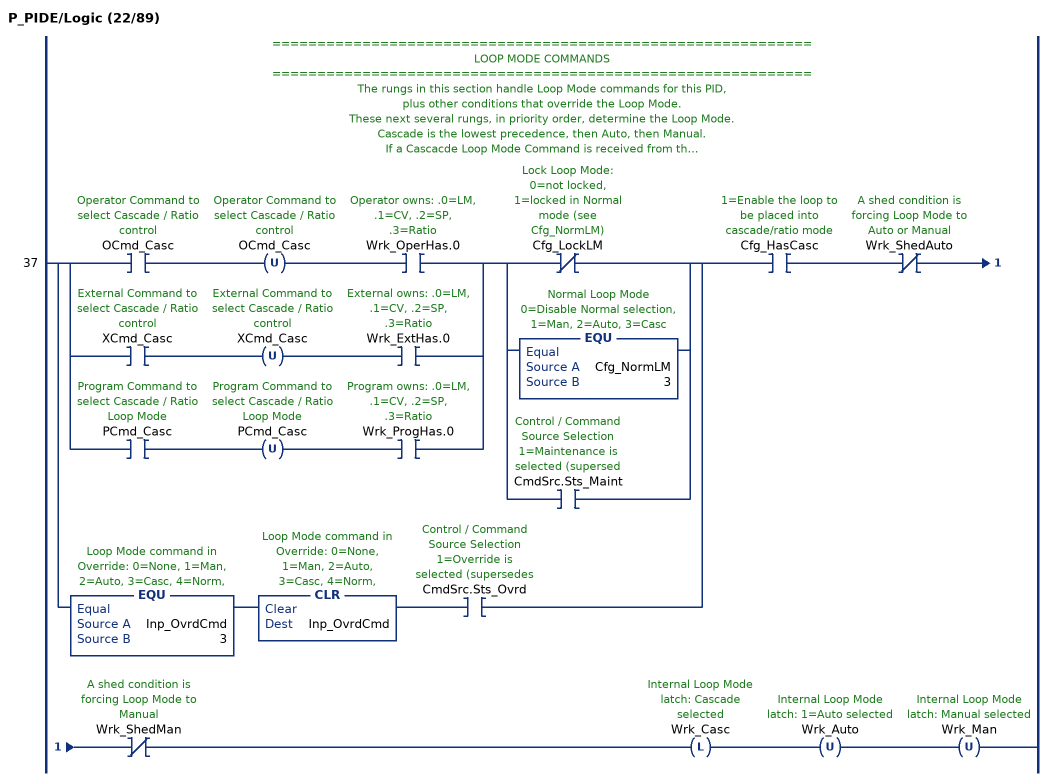
   // ============================================================
   // LOOP MODE COMMANDS
   // ============================================================
   // The rungs in this section handle Loop Mode commands for this PID,
   // plus other conditions that override the Loop Mode.
   // These next several rungs, in priority order, determine the Loop Mode.
   // Cascade is the lowest precedence, then Auto, then Manual.
   // If a Cascacde Loop Mode Command is received from the
   // Loop Mode "owner" (Operator/Maintenance, Program or Override),
   // and if Cascade Loop Mode is permitted, set the Loop Mode to Cascade.
   // #####  V4.00.00 2018-07-16:  Deleted Cfg_PCmdClear. Changed P_Mode to P_CmdSrc.  #####
   // #####  Added External Command Source and Commands.  #####
   37: [[XIC(OCmd_Casc) OTU(OCmd_Casc) XIC(Wrk_OperHas.0) ,XIC(XCmd_Casc) OTU(XCmd_Casc) XIC(Wrk_ExtHas.0) ,XIC(PCmd_Casc) OTU(PCmd_Casc) XIC(Wrk_ProgHas.0) ] [XIO(Cfg_LockLM) ,EQU(Cfg_NormLM,3) ,XIC(CmdSrc.Sts_Maint) ] ,EQU(Inp_OvrdCmd,3) CLR(Inp_OvrdCmd) XIC(CmdSrc.Sts_Ovrd) ]XIC(Cfg_HasCasc)XIO(Wrk_ShedAuto)XIO(Wrk_ShedMan)OTL(Wrk_Casc)OTU(Wrk_Auto)OTU(Wrk_Man);
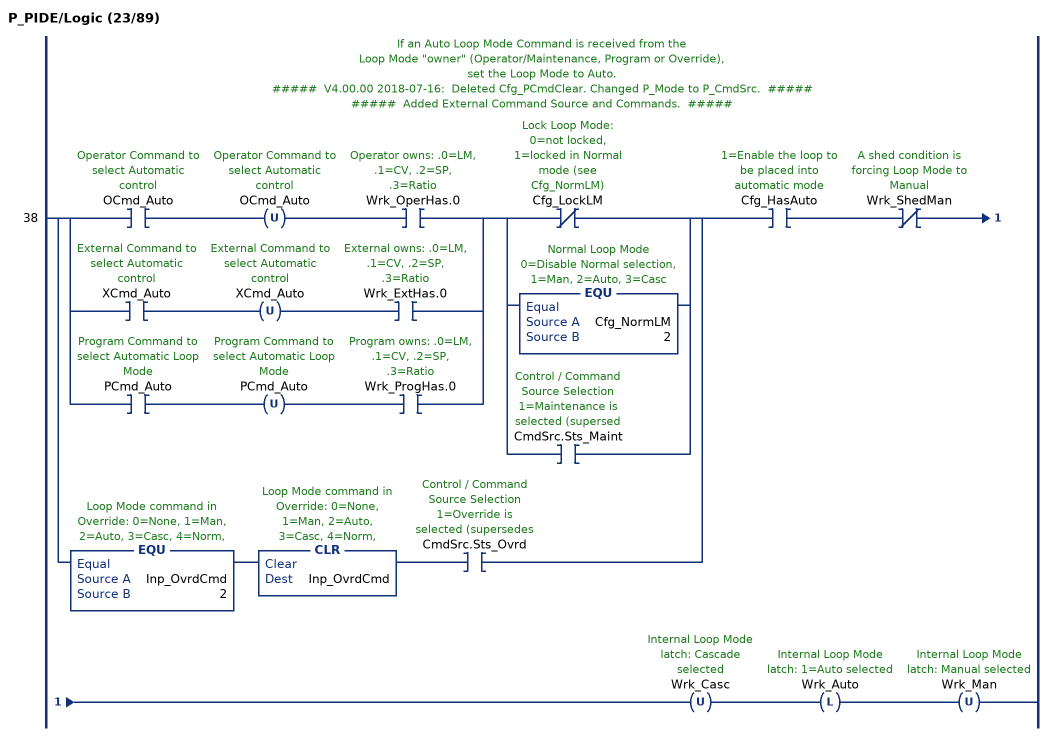
   // If an Auto Loop Mode Command is received from the
   // Loop Mode "owner" (Operator/Maintenance, Program or Override),
   // set the Loop Mode to Auto.
   // #####  V4.00.00 2018-07-16:  Deleted Cfg_PCmdClear. Changed P_Mode to P_CmdSrc.  #####
   // #####  Added External Command Source and Commands.  #####
   38: [[XIC(OCmd_Auto) OTU(OCmd_Auto) XIC(Wrk_OperHas.0) ,XIC(XCmd_Auto) OTU(XCmd_Auto) XIC(Wrk_ExtHas.0) ,XIC(PCmd_Auto) OTU(PCmd_Auto) XIC(Wrk_ProgHas.0) ] [XIO(Cfg_LockLM) ,EQU(Cfg_NormLM,2) ,XIC(CmdSrc.Sts_Maint) ] ,EQU(Inp_OvrdCmd,2) CLR(Inp_OvrdCmd) XIC(CmdSrc.Sts_Ovrd) ]XIC(Cfg_HasAuto)XIO(Wrk_ShedMan)OTU(Wrk_Casc)OTL(Wrk_Auto)OTU(Wrk_Man);
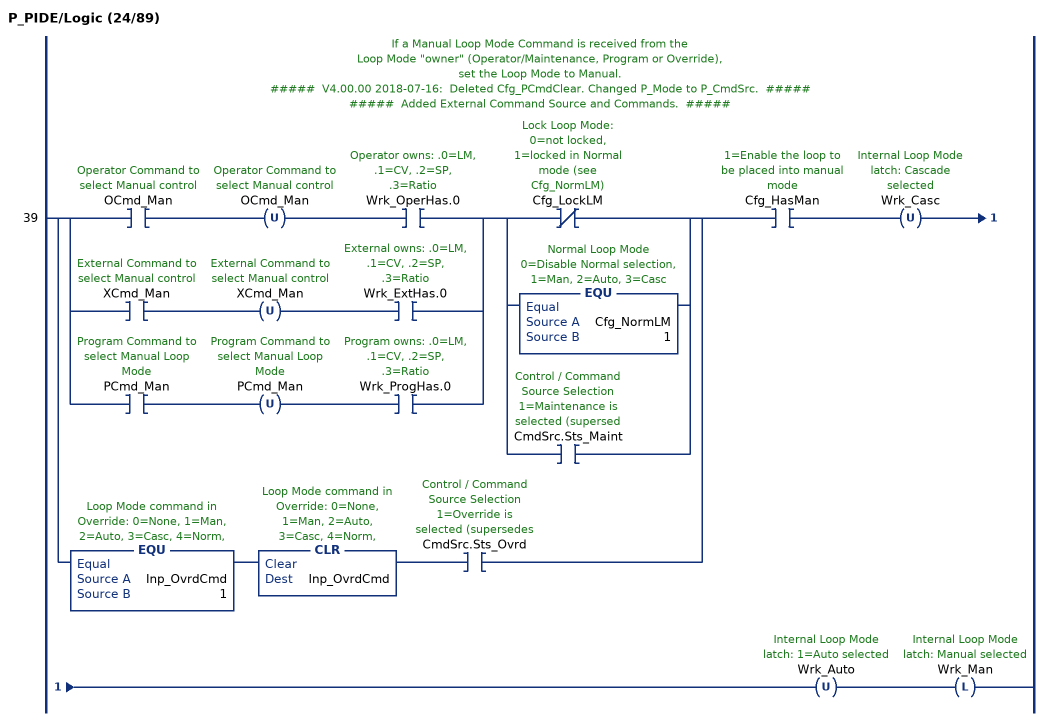
   // If a Manual Loop Mode Command is received from the
   // Loop Mode "owner" (Operator/Maintenance, Program or Override),
   // set the Loop Mode to Manual.
   // #####  V4.00.00 2018-07-16:  Deleted Cfg_PCmdClear. Changed P_Mode to P_CmdSrc.  #####
   // #####  Added External Command Source and Commands.  #####
   39: [[XIC(OCmd_Man) OTU(OCmd_Man) XIC(Wrk_OperHas.0) ,XIC(XCmd_Man) OTU(XCmd_Man) XIC(Wrk_ExtHas.0) ,XIC(PCmd_Man) OTU(PCmd_Man) XIC(Wrk_ProgHas.0) ] [XIO(Cfg_LockLM) ,EQU(Cfg_NormLM,1) ,XIC(CmdSrc.Sts_Maint) ] ,EQU(Inp_OvrdCmd,1) CLR(Inp_OvrdCmd) XIC(CmdSrc.Sts_Ovrd) ]XIC(Cfg_HasMan)OTU(Wrk_Casc)OTU(Wrk_Auto)OTL(Wrk_Man);
